LIN {X 0,Y 572.959,Z 403.806,A -85,B 0,C 180,E1 -2247.187,E2 -2247.187} C_VEL
LIN {X 0,Y 572.946,Z 406.184,A -85,B 0,C 180,E1 -2248.594,E2 -2248.594} C_VEL
LIN {X 0,Y 572.938,Z 407,A -85,B 0,C 180,E1 -2249.999,E2 -2249.999} C_VEL
LIN {X 0,Y 572.946,Z 406.187,A -85,B 0,C 180,E1 -2251.405,E2 -2251.405} C_VEL
LIN {X 0,Y 572.959,Z 403.812,A -85,B 0,C 180,E1 -2252.812,E2 -2252.812} C_VEL
LIN {X 0,Y 573.014,Z 400.898,A -85,B 0,C 180,E1 -2253.867,E2 -2253.867} C_VEL
LIN {X 0,Y 572.963,Z 396.952,A -85,B 0,C 180,E1 -2254.925,E2 -2254.925} C_VEL
LIN {X 0,Y 573.093,Z 391.871,A -85,B 0,C 180,E1 -2255.982,E2 -2255.982} C_VEL
LIN {X 0,Y 573.103,Z 385.474,A -85,B 0,C 180,E1 -2257.043,E2 -2257.043} C_VEL
LIN {X 0,Y 573.177,Z 377.485,A -85,B 0,C 180,E1 -2258.105,E2 -2258.105} C_VEL
LIN {X 0,Y 573.253,Z 369.344,A -85,B 0,C 180,E1 -2258.992,E2 -2258.992} C_VEL
LIN {X 0,Y 573.35,Z 359.411,A -85,B 0,C 180,E1 -2259.88,E2 -2259.88} C_VEL
LIN {X 0,Y 573.523,Z 348.2,A -85,B 0,C 180,E1 -2260.68,E2 -2260.68} C_VEL
LIN {X 0,Y 573.627,Z 337.193,A -85,B 0,C 180,E1 -2261.304,E2 -2261.304} C_VEL
LIN {X 0,Y 573.704,Z 325.004,A -85,B 0,C 180,E1 -2261.84,E2 -2261.84} C_VEL
LIN {X 0,Y 573.831,Z 312.213,A -85,B 0,C 180,E1 -2262.241,E2 -2262.241} C_VEL
LIN {X 0,Y 573.922,Z 298.664,A -85,B 0,C 180,E1 -2262.508,E2 -2262.508} C_VEL
LIN {X 0,Y 574.023,Z 199.578,A -85,B 0,C 180,E1 -2263.757,E2 -2263.757} C_VEL
LIN {X 0,Y 573.377,Z 195.275,A -85,B 0,C 180,E1 -2263.85,E2 -2263.85} C_VEL
LIN {X 0,Y 573.52,Z 177.034,A -85,B 0,C 180,E1 -2266.545,E2 -2266.545} C_VEL
LIN {X 0,Y 573.652,Z 159.914,A -85,B 0,C 180,E1 -2269.13,E2 -2269.13} C_VEL
LIN {X 0,Y 573.855,Z 142.746,A -85,B 0,C 180,E1 -2271.744,E2 -2271.744} C_VEL
LIN {X 0,Y 573.214,Z 138.649,A -85,B 0,C 180,E1 -2272.433,E2 -2272.433} C_VEL
LIN {X 0,Y 573.225,Z 138.584,A -85,B 0,C 180,E1 -2275.41,E2 -2275.41} C_VEL
LIN {X 0,Y 573.186,Z 138.585,A -85,B 0,C 180,E1 -2278.016,E2 -2278.016} C_VEL
LIN {X 0,Y 573.201,Z 138.581,A -85,B 0,C 180,E1 -2280.877,E2 -2280.877} C_VEL
LIN {X 0,Y 573.237,Z 138.584,A -85,B 0,C 180,E1 -2283.519,E2 -2283.519} C_VEL
LIN {X 0,Y 573.177,Z 138.584,A -85,B 0,C 180,E1 -2286.053,E2 -2286.053} C_VEL
LIN {X 0,Y 573.17,Z 138.584,A -85,B 0,C 180,E1 -2288.706,E2 -2288.706} C_VEL
LIN {X 0,Y 573.194,Z 138.589,A -85,B 0,C 180,E1 -2291.459,E2 -2291.459} C_VEL
LIN {X 0,Y 573.196,Z 138.58,A -85,B 0,C 180,E1 -2294.335,E2 -2294.335} C_VEL
LIN {X 0,Y 573.189,Z 138.582,A -85,B 0,C 180,E1 -2296.636,E2 -2296.636} C_VEL
LIN {X 0,Y 573.236,Z 138.581,A -85,B 0,C 180,E1 -2299.474,E2 -2299.474} C_VEL
LIN {X 0,Y 573.205,Z 138.578,A -85,B 0,C 180,E1 -2302.19,E2 -2302.19} C_VEL
LIN {X 0,Y 573.215,Z 138.586,A -85,B 0,C 180,E1 -2305.229,E2 -2305.229} C_VEL
LIN {X 0,Y 573.218,Z 138.578,A -85,B 0,C 180,E1 -2307.774,E2 -2307.774} C_VEL
LIN {X 0,Y 573.218,Z 138.58,A -85,B 0,C 180,E1 -2310.631,E2 -2310.631} C_VEL
LIN {X 0,Y 573.189,Z 138.583,A -85,B 0,C 180,E1 -2313.514,E2 -2313.514} C_VEL
LIN {X 0,Y 573.18,Z 138.582,A -85,B 0,C 180,E1 -2316.132,E2 -2316.132} C_VEL
LIN {X 0,Y 573.23,Z 138.581,A -85,B 0,C 180,E1 -2319.173,E2 -2319.173} C_VEL
LIN {X 0,Y 573.189,Z 138.582,A -85,B 0,C 180,E1 -2321.41,E2 -2321.41} C_VEL
LIN {X 0,Y 573.211,Z 138.578,A -85,B 0,C 180,E1 -2323.62,E2 -2323.62} C_VEL
LIN {X 0,Y 573.187,Z 138.586,A -85,B 0,C 180,E1 -2326.528,E2 -2326.528} C_VEL
LIN {X 0,Y 573.221,Z 138.577,A -85,B 0,C 180,E1 -2329.402,E2 -2329.402} C_VEL
LIN {X 0,Y 573.245,Z 138.577,A -85,B 0,C 180,E1 -2332.249,E2 -2332.249} C_VEL
LIN {X 0,Y 573.269,Z 138.574,A -85,B 0,C 180,E1 -2335.077,E2 -2335.077} C_VEL
LIN {X 0,Y 573.27,Z 138.571,A -85,B 0,C 180,E1 -2337.892,E2 -2337.892} C_VEL
LIN {X 0,Y 573.317,Z 138.572,A -85,B 0,C 180,E1 -2340.702,E2 -2340.702} C_VEL
LIN {X 0,Y 573.281,Z 138.574,A -85,B 0,C 180,E1 -2342.81,E2 -2342.81} C_VEL
LIN {X 0,Y 573.246,Z 138.574,A -85,B 0,C 180,E1 -2345.628,E2 -2345.628} C_VEL
LIN {X 0,Y 573.197,Z 138.581,A -85,B 0,C 180,E1 -2347.751,E2 -2347.751} C_VEL
LIN {X 0,Y 573.225,Z 138.583,A -85,B 0,C 180,E1 -2350.597,E2 -2350.597} C_VEL
LIN {X 0,Y 573.194,Z 138.58,A -85,B 0,C 180,E1 -2353.471,E2 -2353.471} C_VEL
LIN {X 0,Y 573.197,Z 138.581,A -85,B 0,C 180,E1 -2355.649,E2 -2355.649} C_VEL
LIN {X 0,Y 573.192,Z 138.584,A -85,B 0,C 180,E1 -2357.85,E2 -2357.85} C_VEL
LIN {X 0,Y 573.218,Z 138.585,A -85,B 0,C 180,E1 -2360.077,E2 -2360.077} C_VEL
LIN {X 0,Y 573.212,Z 138.586,A -85,B 0,C 180,E1 -2362.338,E2 -2362.338} C_VEL
LIN {X 0,Y 573.2,Z 138.581,A -85,B 0,C 180,E1 -2364.394,E2 -2364.394} C_VEL
LIN {X 0,Y 572.557,Z 138.663,A -85,B 0,C 180,E1 -2364.98,E2 -2364.98} C_VEL
LIN {X 0,Y 569.712,Z 139.02,A -85,B 0,C 180,E1 -2365.932,E2 -2365.932} C_VEL
LIN {X 0,Y 567.284,Z 139.319,A -85,B 0,C 180,E1 -2366.697,E2 -2366.697} C_VEL
LIN {X 0,Y 566.228,Z 139.449,A -85,B 0,C 180,E1 -2367.288,E2 -2367.288} C_VEL
LIN {X 0,Y 566.136,Z 139.461,A -85,B 0,C 180,E1 -2367.489,E2 -2367.489} C_VEL
LIN {X 0,Y 566.152,Z 139.462,A -85,B 0,C 180,E1 -2370.594,E2 -2370.594} C_VEL
LIN {X 0,Y 566.246,Z 139.591,A -85,B 0,C 180,E1 -2373.411,E2 -2373.411} C_VEL
LIN {X 0,Y 566.641,Z 143.669,A -85,B 0,C 180,E1 -2374.141,E2 -2374.141} C_VEL
LIN {X 0,Y 566.474,Z 160.639,A -85,B 0,C 180,E1 -2376.988,E2 -2376.988} C_VEL
LIN {X 0,Y 566.291,Z 178.737,A -85,B 0,C 180,E1 -2380,E2 -2380} C_VEL
LIN {X 0,Y 566.525,Z 180.469,A -85,B 0,C 180,E1 -2380.076,E2 -2380.076} C_VEL
LIN {X 0,Y 567.177,Z 186.806,A -85,B 0,C 180,E1 -2380.173,E2 -2380.173} C_VEL
LIN {X 0,Y 566.986,Z 285.959,A -85,B 0,C 180,E1 -2381.451,E2 -2381.451} C_VEL
LIN {X 0,Y 566.852,Z 298.233,A -85,B 0,C 180,E1 -2381.738,E2 -2381.738} C_VEL
LIN {X 0,Y 566.78,Z 308.773,A -85,B 0,C 180,E1 -2382.095,E2 -2382.095} C_VEL
LIN {X 0,Y 566.656,Z 318.628,A -85,B 0,C 180,E1 -2382.527,E2 -2382.527} C_VEL
LIN {X 0,Y 566.545,Z 328.715,A -85,B 0,C 180,E1 -2383.082,E2 -2383.082} C_VEL
LIN {X 0,Y 566.369,Z 338.546,A -85,B 0,C 180,E1 -2383.747,E2 -2383.747} C_VEL
LIN {X 0,Y 566.28,Z 348.816,A -85,B 0,C 180,E1 -2384.598,E2 -2384.598} C_VEL
LIN {X 0,Y 566.11,Z 358.337,A -85,B 0,C 180,E1 -2385.585,E2 -2385.585} C_VEL
LIN {X 0,Y 566.05,Z 365.537,A -85,B 0,C 180,E1 -2386.497,E2 -2386.497} C_VEL
LIN {X 0,Y 565.975,Z 372.063,A -85,B 0,C 180,E1 -2387.498,E2 -2387.498} C_VEL
LIN {X 0,Y 565.954,Z 377.399,A -85,B 0,C 180,E1 -2388.503,E2 -2388.503} C_VEL
LIN {X 0,Y 565.92,Z 382.712,A -85,B 0,C 180,E1 -2389.778,E2 -2389.778} C_VEL
LIN {X 0,Y 565.842,Z 385.534,A -85,B 0,C 180,E1 -2390.697,E2 -2390.697} C_VEL
LIN {X 0,Y 565.844,Z 387.622,A -85,B 0,C 180,E1 -2391.611,E2 -2391.611} C_VEL
LIN {X 0,Y 565.828,Z 389.187,A -85,B 0,C 180,E1 -2392.648,E2 -2392.648} C_VEL
LIN {X 0,Y 565.813,Z 389.96,A -85,B 0,C 180,E1 -2393.839,E2 -2393.839} C_VEL
LIN {X 0,Y 565.849,Z 389.512,A -85,B 0,C 180,E1 -2395.158,E2 -2395.158} C_VEL
LIN {X 0,Y 565.86,Z 387.946,A -85,B 0,C 180,E1 -2396.319,E2 -2396.319} C_VEL
LIN {X 0,Y 565.883,Z 384.566,A -85,B 0,C 180,E1 -2397.723,E2 -2397.723} C_VEL
LIN {X 0,Y 565.936,Z 381.748,A -85,B 0,C 180,E1 -2398.564,E2 -2398.564} C_VEL
LIN {X 0,Y 565.945,Z 376.347,A -85,B 0,C 180,E1 -2399.807,E2 -2399.807} C_VEL
LIN {X 0,Y 566.013,Z 369.386,A -85,B 0,C 180,E1 -2401.038,E2 -2401.038} C_VEL
LIN {X 0,Y 566.097,Z 362.063,A -85,B 0,C 180,E1 -2402.054,E2 -2402.054} C_VEL
LIN {X 0,Y 566.182,Z 355.241,A -85,B 0,C 180,E1 -2402.847,E2 -2402.847} C_VEL
LIN {X 0,Y 566.273,Z 346.877,A -85,B 0,C 180,E1 -2403.662,E2 -2403.662} C_VEL
LIN {X 0,Y 566.371,Z 338.436,A -85,B 0,C 180,E1 -2404.351,E2 -2404.351} C_VEL
LIN {X 0,Y 566.495,Z 329.013,A -85,B 0,C 180,E1 -2404.99,E2 -2404.99} C_VEL
LIN {X 0,Y 566.641,Z 318.934,A -85,B 0,C 180,E1 -2405.548,E2 -2405.548} C_VEL
LIN {X 0,Y 566.78,Z 307.631,A -85,B 0,C 180,E1 -2406.042,E2 -2406.042} C_VEL
LIN {X 0,Y 566.903,Z 293.652,A -85,B 0,C 180,E1 -2406.476,E2 -2406.476} C_VEL
LIN {X 0,Y 566.983,Z 281.874,A -85,B 0,C 180,E1 -2406.705,E2 -2406.705} C_VEL
LIN {X 0,Y 567.054,Z 183.818,A -85,B 0,C 180,E1 -2407.958,E2 -2407.958} C_VEL
LIN {X 0,Y 566.338,Z 179.288,A -85,B 0,C 180,E1 -2408.049,E2 -2408.049} C_VEL
LIN {X 0,Y 566.292,Z 178.336,A -85,B 0,C 180,E1 -2408.143,E2 -2408.143} C_VEL
LIN {X 0,Y 566.417,Z 162.116,A -85,B 0,C 180,E1 -2410.872,E2 -2410.872} C_VEL
LIN {X 0,Y 566.688,Z 143.921,A -85,B 0,C 180,E1 -2413.983,E2 -2413.983} C_VEL
LIN {X 0,Y 566.248,Z 139.507,A -85,B 0,C 180,E1 -2414.801,E2 -2414.801} C_VEL
LIN {X 0,Y 566.24,Z 139.454,A -85,B 0,C 180,E1 -2417.82,E2 -2417.82} C_VEL
LIN {X 0,Y 566.209,Z 139.451,A -85,B 0,C 180,E1 -2420.715,E2 -2420.715} C_VEL
LIN {X 0,Y 566.262,Z 139.444,A -85,B 0,C 180,E1 -2423.164,E2 -2423.164} C_VEL
LIN {X 0,Y 566.182,Z 139.461,A -85,B 0,C 180,E1 -2425.73,E2 -2425.73} C_VEL
LIN {X 0,Y 566.275,Z 139.451,A -85,B 0,C 180,E1 -2427.867,E2 -2427.867} C_VEL
LIN {X 0,Y 566.298,Z 139.439,A -85,B 0,C 180,E1 -2430.712,E2 -2430.712} C_VEL
LIN {X 0,Y 566.268,Z 139.443,A -85,B 0,C 180,E1 -2432.846,E2 -2432.846} C_VEL
LIN {X 0,Y 566.254,Z 139.453,A -85,B 0,C 180,E1 -2435.699,E2 -2435.699} C_VEL
LIN {X 0,Y 566.204,Z 139.451,A -85,B 0,C 180,E1 -2438.567,E2 -2438.567} C_VEL
LIN {X 0,Y 566.241,Z 139.455,A -85,B 0,C 180,E1 -2441.455,E2 -2441.455} C_VEL
LIN {X 0,Y 566.228,Z 139.448,A -85,B 0,C 180,E1 -2444.505,E2 -2444.505} C_VEL
LIN {X 0,Y 566.198,Z 139.461,A -85,B 0,C 180,E1 -2447.332,E2 -2447.332} C_VEL
LIN {X 0,Y 566.206,Z 139.45,A -85,B 0,C 180,E1 -2450.338,E2 -2450.338} C_VEL
LIN {X 0,Y 566.17,Z 139.464,A -85,B 0,C 180,E1 -2453.282,E2 -2453.282} C_VEL
LIN {X 0,Y 566.207,Z 139.452,A -85,B 0,C 180,E1 -2455.75,E2 -2455.75} C_VEL
LIN {X 0,Y 566.202,Z 139.451,A -85,B 0,C 180,E1 -2458.202,E2 -2458.202} C_VEL
LIN {X 0,Y 566.185,Z 139.463,A -85,B 0,C 180,E1 -2461.076,E2 -2461.076} C_VEL
LIN {X 0,Y 566.196,Z 139.452,A -85,B 0,C 180,E1 -2463.732,E2 -2463.732} C_VEL
LIN {X 0,Y 566.198,Z 139.455,A -85,B 0,C 180,E1 -2466.57,E2 -2466.57} C_VEL
LIN {X 0,Y 566.211,Z 139.45,A -85,B 0,C 180,E1 -2469.686,E2 -2469.686} C_VEL
LIN {X 0,Y 566.197,Z 139.46,A -85,B 0,C 180,E1 -2472.917,E2 -2472.917} C_VEL
LIN {X 0,Y 566.192,Z 139.453,A -85,B 0,C 180,E1 -2476.05,E2 -2476.05} C_VEL
LIN {X 0,Y 566.201,Z 139.453,A -85,B 0,C 180,E1 -2479.215,E2 -2479.215} C_VEL
LIN {X 0,Y 566.179,Z 139.454,A -85,B 0,C 180,E1 -2481.637,E2 -2481.637} C_VEL
LIN {X 0,Y 566.147,Z 139.463,A -85,B 0,C 180,E1 -2484.307,E2 -2484.307} C_VEL
LIN {X 0,Y 566.217,Z 139.453,A -85,B 0,C 180,E1 -2486.898,E2 -2486.898} C_VEL
LIN {X 0,Y 566.174,Z 139.454,A -85,B 0,C 180,E1 -2489.407,E2 -2489.407} C_VEL
LIN {X 0,Y 566.185,Z 139.455,A -85,B 0,C 180,E1 -2491.856,E2 -2491.856} C_VEL
LIN {X 0,Y 566.236,Z 139.447,A -85,B 0,C 180,E1 -2495.039,E2 -2495.039} C_VEL
LIN {X 0,Y 566.184,Z 139.461,A -85,B 0,C 180,E1 -2498.137,E2 -2498.137} C_VEL
LIN {X 0,Y 566.229,Z 139.451,A -85,B 0,C 180,E1 -2500.614,E2 -2500.614} C_VEL
LIN {X 0,Y 566.176,Z 139.455,A -85,B 0,C 180,E1 -2503.412,E2 -2503.412} C_VEL
LIN {X 0,Y 566.181,Z 139.459,A -85,B 0,C 180,E1 -2506.359,E2 -2506.359} C_VEL
LIN {X 0,Y 566.234,Z 139.448,A -85,B 0,C 180,E1 -2508.676,E2 -2508.676} C_VEL
LIN {X 0,Y 566.198,Z 139.454,A -85,B 0,C 180,E1 -2511.434,E2 -2511.434} C_VEL
LIN {X 0,Y 566.235,Z 139.45,A -85,B 0,C 180,E1 -2514.302,E2 -2514.302} C_VEL
LIN {X 0,Y 566.271,Z 139.452,A -85,B 0,C 180,E1 -2517.867,E2 -2517.867} C_VEL
LIN {X 0,Y 566.279,Z 139.448,A -85,B 0,C 180,E1 -2520,E2 -2520} C_VEL
LIN {X 0,Y 566.249,Z 139.445,A -85,B 0,C 180,E1 -2522.846,E2 -2522.846} C_VEL
LIN {X 0,Y 566.24,Z 139.456,A -85,B 0,C 180,E1 -2525.699,E2 -2525.699} C_VEL
LIN {X 0,Y 566.187,Z 139.453,A -85,B 0,C 180,E1 -2528.567,E2 -2528.567} C_VEL
LIN {X 0,Y 566.238,Z 139.455,A -85,B 0,C 180,E1 -2531.455,E2 -2531.455} C_VEL
LIN {X 0,Y 566.176,Z 139.454,A -85,B 0,C 180,E1 -2534.483,E2 -2534.483} C_VEL
LIN {X 0,Y 566.181,Z 139.462,A -85,B 0,C 180,E1 -2537.333,E2 -2537.333} C_VEL
LIN {X 0,Y 566.196,Z 139.458,A -85,B 0,C 180,E1 -2539.581,E2 -2539.581} C_VEL
LIN {X 0,Y 566.181,Z 139.455,A -85,B 0,C 180,E1 -2541.863,E2 -2541.863} C_VEL
LIN {X 0,Y 566.152,Z 139.457,A -85,B 0,C 180,E1 -2544.183,E2 -2544.183} C_VEL
LIN {X 0,Y 566.166,Z 139.457,A -85,B 0,C 180,E1 -2546.651,E2 -2546.651} C_VEL
LIN {X 0,Y 566.146,Z 139.459,A -85,B 0,C 180,E1 -2549.772,E2 -2549.772} C_VEL
LIN {X 0,Y 566.176,Z 139.455,A -85,B 0,C 180,E1 -2552.425,E2 -2552.425} C_VEL
LIN {X 0,Y 566.164,Z 139.465,A -85,B 0,C 180,E1 -2554.987,E2 -2554.987} C_VEL
LIN {X 0,Y 566.185,Z 139.456,A -85,B 0,C 180,E1 -2557.462,E2 -2557.462} C_VEL
LIN {X 0,Y 566.159,Z 139.457,A -85,B 0,C 180,E1 -2560.204,E2 -2560.204} C_VEL
LIN {X 0,Y 566.144,Z 139.464,A -85,B 0,C 180,E1 -2563.06,E2 -2563.06} C_VEL
LIN {X 0,Y 566.144,Z 139.459,A -85,B 0,C 180,E1 -2566.055,E2 -2566.055} C_VEL
LIN {X 0,Y 566.138,Z 139.466,A -85,B 0,C 180,E1 -2568.857,E2 -2568.857} C_VEL
LIN {X 0,Y 566.13,Z 139.46,A -85,B 0,C 180,E1 -2571.453,E2 -2571.453} C_VEL
LIN {X 0,Y 566.152,Z 139.457,A -85,B 0,C 180,E1 -2573.793,E2 -2573.793} C_VEL
LIN {X 0,Y 566.143,Z 139.462,A -85,B 0,C 180,E1 -2576.892,E2 -2576.892} C_VEL
LIN {X 0,Y 566.149,Z 139.458,A -85,B 0,C 180,E1 -2579.405,E2 -2579.405} C_VEL
LIN {X 0,Y 566.133,Z 139.462,A -85,B 0,C 180,E1 -2581.853,E2 -2581.853} C_VEL
LIN {X 0,Y 566.178,Z 139.462,A -85,B 0,C 180,E1 -2584.249,E2 -2584.249} C_VEL
LIN {X 0,Y 566.178,Z 139.567,A -85,B 0,C 180,E1 -2587.416,E2 -2587.416} C_VEL
LIN {X 0,Y 566.945,Z 143.998,A -85,B 0,C 180,E1 -2588.167,E2 -2588.167} C_VEL
LIN {X 0,Y 566.702,Z 161.238,A -85,B 0,C 180,E1 -2590.837,E2 -2590.837} C_VEL
LIN {X 0,Y 566.514,Z 177.105,A -85,B 0,C 180,E1 -2593.261,E2 -2593.261} C_VEL
LIN {X 0,Y 566.384,Z 195.262,A -85,B 0,C 180,E1 -2595.974,E2 -2595.974} C_VEL
LIN {X 0,Y 567.129,Z 200.463,A -85,B 0,C 180,E1 -2596.084,E2 -2596.084} C_VEL
LIN {X 0,Y 566.982,Z 302.917,A -85,B 0,C 180,E1 -2597.403,E2 -2597.403} C_VEL
LIN {X 0,Y 566.858,Z 316.198,A -85,B 0,C 180,E1 -2597.718,E2 -2597.718} C_VEL
LIN {X 0,Y 566.73,Z 328.363,A -85,B 0,C 180,E1 -2598.147,E2 -2598.147} C_VEL
LIN {X 0,Y 566.629,Z 340.142,A -85,B 0,C 180,E1 -2598.708,E2 -2598.708} C_VEL
LIN {X 0,Y 566.461,Z 352.187,A -85,B 0,C 180,E1 -2599.455,E2 -2599.455} C_VEL
LIN {X 0,Y 566.326,Z 362.597,A -85,B 0,C 180,E1 -2600.265,E2 -2600.265} C_VEL
LIN {X 0,Y 566.207,Z 371.107,A -85,B 0,C 180,E1 -2601.074,E2 -2601.074} C_VEL
LIN {X 0,Y 566.113,Z 378.955,A -85,B 0,C 180,E1 -2601.971,E2 -2601.971} C_VEL
LIN {X 0,Y 566.004,Z 386.619,A -85,B 0,C 180,E1 -2603.046,E2 -2603.046} C_VEL
LIN {X 0,Y 566.004,Z 393.676,A -85,B 0,C 180,E1 -2604.298,E2 -2604.298} C_VEL
LIN {X 0,Y 565.933,Z 398.37,A -85,B 0,C 180,E1 -2605.369,E2 -2605.369} C_VEL
LIN {X 0,Y 565.927,Z 401.956,A -85,B 0,C 180,E1 -2606.439,E2 -2606.439} C_VEL
LIN {X 0,Y 565.878,Z 403.806,A -85,B 0,C 180,E1 -2607.152,E2 -2607.152} C_VEL
LIN {X 0,Y 565.846,Z 406.183,A -85,B 0,C 180,E1 -2608.576,E2 -2608.576} C_VEL
LIN {X 0,Y 565.839,Z 407,A -85,B 0,C 180,E1 -2609.999,E2 -2609.999} C_VEL
LIN {X 0,Y 565.846,Z 406.186,A -85,B 0,C 180,E1 -2611.423,E2 -2611.423} C_VEL
LIN {X 0,Y 565.878,Z 403.812,A -85,B 0,C 180,E1 -2612.847,E2 -2612.847} C_VEL
LIN {X 0,Y 565.926,Z 400.898,A -85,B 0,C 180,E1 -2613.916,E2 -2613.916} C_VEL
LIN {X 0,Y 565.878,Z 396.952,A -85,B 0,C 180,E1 -2614.987,E2 -2614.987} C_VEL
LIN {X 0,Y 566.004,Z 391.872,A -85,B 0,C 180,E1 -2616.058,E2 -2616.058} C_VEL
LIN {X 0,Y 566.039,Z 385.473,A -85,B 0,C 180,E1 -2617.131,E2 -2617.131} C_VEL
LIN {X 0,Y 566.133,Z 377.485,A -85,B 0,C 180,E1 -2618.207,E2 -2618.207} C_VEL
LIN {X 0,Y 566.228,Z 369.343,A -85,B 0,C 180,E1 -2619.105,E2 -2619.105} C_VEL
LIN {X 0,Y 566.351,Z 359.409,A -85,B 0,C 180,E1 -2620.004,E2 -2620.004} C_VEL
LIN {X 0,Y 566.544,Z 348.298,A -85,B 0,C 180,E1 -2620.806,E2 -2620.806} C_VEL
LIN {X 0,Y 566.659,Z 337.191,A -85,B 0,C 180,E1 -2621.445,E2 -2621.445} C_VEL
LIN {X 0,Y 566.743,Z 325.002,A -85,B 0,C 180,E1 -2621.987,E2 -2621.987} C_VEL
LIN {X 0,Y 566.907,Z 312.212,A -85,B 0,C 180,E1 -2622.393,E2 -2622.393} C_VEL
LIN {X 0,Y 567,Z 300.167,A -85,B 0,C 180,E1 -2622.641,E2 -2622.641} C_VEL
LIN {X 0,Y 567.039,Z 199.902,A -85,B 0,C 180,E1 -2623.925,E2 -2623.925} C_VEL
LIN {X 0,Y 566.37,Z 195.286,A -85,B 0,C 180,E1 -2624.025,E2 -2624.025} C_VEL
LIN {X 0,Y 566.53,Z 176.033,A -85,B 0,C 180,E1 -2626.896,E2 -2626.896} C_VEL
LIN {X 0,Y 566.715,Z 158.543,A -85,B 0,C 180,E1 -2629.561,E2 -2629.561} C_VEL
LIN {X 0,Y 566.892,Z 143.82,A -85,B 0,C 180,E1 -2631.833,E2 -2631.833} C_VEL
LIN {X 0,Y 566.189,Z 139.553,A -85,B 0,C 180,E1 -2632.558,E2 -2632.558} C_VEL
LIN {X 0,Y 566.186,Z 139.462,A -85,B 0,C 180,E1 -2635.749,E2 -2635.749} C_VEL
LIN {X 0,Y 566.131,Z 139.463,A -85,B 0,C 180,E1 -2638.188,E2 -2638.188} C_VEL
LIN {X 0,Y 566.17,Z 139.459,A -85,B 0,C 180,E1 -2641.072,E2 -2641.072} C_VEL
LIN {X 0,Y 566.19,Z 139.459,A -85,B 0,C 180,E1 -2643.73,E2 -2643.73} C_VEL
LIN {X 0,Y 566.137,Z 139.46,A -85,B 0,C 180,E1 -2646.573,E2 -2646.573} C_VEL
LIN {X 0,Y 566.192,Z 139.458,A -85,B 0,C 180,E1 -2649.683,E2 -2649.683} C_VEL
LIN {X 0,Y 566.141,Z 139.462,A -85,B 0,C 180,E1 -2652.91,E2 -2652.91} C_VEL
LIN {X 0,Y 566.144,Z 139.459,A -85,B 0,C 180,E1 -2656.053,E2 -2656.053} C_VEL
LIN {X 0,Y 566.144,Z 139.462,A -85,B 0,C 180,E1 -2658.857,E2 -2658.857} C_VEL
LIN {X 0,Y 566.188,Z 139.458,A -85,B 0,C 180,E1 -2661.443,E2 -2661.443} C_VEL
LIN {X 0,Y 566.132,Z 139.46,A -85,B 0,C 180,E1 -2664.305,E2 -2664.305} C_VEL
LIN {X 0,Y 566.15,Z 139.463,A -85,B 0,C 180,E1 -2666.893,E2 -2666.893} C_VEL
LIN {X 0,Y 566.147,Z 139.462,A -85,B 0,C 180,E1 -2669.405,E2 -2669.405} C_VEL
LIN {X 0,Y 566.138,Z 139.459,A -85,B 0,C 180,E1 -2671.853,E2 -2671.853} C_VEL
LIN {X 0,Y 566.169,Z 139.456,A -85,B 0,C 180,E1 -2674.249,E2 -2674.249} C_VEL
LIN {X 0,Y 566.146,Z 139.461,A -85,B 0,C 180,E1 -2677.367,E2 -2677.367} C_VEL
LIN {X 0,Y 566.185,Z 139.453,A -85,B 0,C 180,E1 -2679.661,E2 -2679.661} C_VEL
LIN {X 0,Y 566.161,Z 139.456,A -85,B 0,C 180,E1 -2681.92,E2 -2681.92} C_VEL
LIN {X 0,Y 566.169,Z 139.463,A -85,B 0,C 180,E1 -2684.889,E2 -2684.889} C_VEL
LIN {X 0,Y 566.163,Z 139.456,A -85,B 0,C 180,E1 -2687.817,E2 -2687.817} C_VEL
LIN {X 0,Y 566.141,Z 139.459,A -85,B 0,C 180,E1 -2689.991,E2 -2689.991} C_VEL
LIN {X 0,Y 566.225,Z 139.454,A -85,B 0,C 180,E1 -2692.87,E2 -2692.87} C_VEL
LIN {X 0,Y 566.245,Z 139.449,A -85,B 0,C 180,E1 -2695.015,E2 -2695.015} C_VEL
LIN {X 0,Y 566.244,Z 139.446,A -85,B 0,C 180,E1 -2697.866,E2 -2697.866} C_VEL
LIN {X 0,Y 566.286,Z 139.448,A -85,B 0,C 180,E1 -2700.711,E2 -2700.711} C_VEL
LIN {X 0,Y 566.245,Z 139.449,A -85,B 0,C 180,E1 -2702.845,E2 -2702.845} C_VEL
LIN {X 0,Y 566.217,Z 139.45,A -85,B 0,C 180,E1 -2705.698,E2 -2705.698} C_VEL
LIN {X 0,Y 566.168,Z 139.457,A -85,B 0,C 180,E1 -2707.848,E2 -2707.848} C_VEL
LIN {X 0,Y 566.195,Z 139.456,A -85,B 0,C 180,E1 -2710.73,E2 -2710.73} C_VEL
LIN {X 0,Y 566.163,Z 139.458,A -85,B 0,C 180,E1 -2712.911,E2 -2712.911} C_VEL
LIN {X 0,Y 566.17,Z 139.456,A -85,B 0,C 180,E1 -2715.11,E2 -2715.11} C_VEL
LIN {X 0,Y 566.153,Z 139.464,A -85,B 0,C 180,E1 -2718.079,E2 -2718.079} C_VEL
LIN {X 0,Y 566.186,Z 139.461,A -85,B 0,C 180,E1 -2720.338,E2 -2720.338} C_VEL
LIN {X 0,Y 566.151,Z 139.458,A -85,B 0,C 180,E1 -2723.28,E2 -2723.28} C_VEL
LIN {X 0,Y 566.172,Z 139.459,A -85,B 0,C 180,E1 -2725.751,E2 -2725.751} C_VEL
LIN {X 0,Y 566.136,Z 139.461,A -85,B 0,C 180,E1 -2727.489,E2 -2727.489} C_VEL
LIN {X 0,Y 565.452,Z 139.554,A -85,B 0,C 180,E1 -2728.082,E2 -2728.082} C_VEL
LIN {X 0,Y 562.596,Z 139.908,A -85,B 0,C 180,E1 -2729.046,E2 -2729.046} C_VEL
LIN {X 0,Y 560.202,Z 140.206,A -85,B 0,C 180,E1 -2729.822,E2 -2729.822} C_VEL
LIN {X 0,Y 559.187,Z 140.332,A -85,B 0,C 180,E1 -2730.421,E2 -2730.421} C_VEL
LIN {X 0,Y 559.11,Z 140.338,A -85,B 0,C 180,E1 -2730.624,E2 -2730.624} C_VEL
LIN {X 0,Y 559.184,Z 140.438,A -85,B 0,C 180,E1 -2733.303,E2 -2733.303} C_VEL
LIN {X 0,Y 559.641,Z 144.369,A -85,B 0,C 180,E1 -2734.024,E2 -2734.024} C_VEL
LIN {X 0,Y 559.477,Z 160.467,A -85,B 0,C 180,E1 -2736.754,E2 -2736.754} C_VEL
LIN {X 0,Y 559.283,Z 179.019,A -85,B 0,C 180,E1 -2739.842,E2 -2739.842} C_VEL
LIN {X 0,Y 560.263,Z 185.188,A -85,B 0,C 180,E1 -2739.977,E2 -2739.977} C_VEL
LIN {X 0,Y 560.037,Z 285.586,A -85,B 0,C 180,E1 -2741.287,E2 -2741.287} C_VEL
LIN {X 0,Y 559.926,Z 298.604,A -85,B 0,C 180,E1 -2741.596,E2 -2741.596} C_VEL
LIN {X 0,Y 559.811,Z 309.088,A -85,B 0,C 180,E1 -2741.958,E2 -2741.958} C_VEL
LIN {X 0,Y 559.732,Z 317.871,A -85,B 0,C 180,E1 -2742.345,E2 -2742.345} C_VEL
LIN {X 0,Y 559.578,Z 327.966,A -85,B 0,C 180,E1 -2742.898,E2 -2742.898} C_VEL
LIN {X 0,Y 559.404,Z 336.205,A -85,B 0,C 180,E1 -2743.444,E2 -2743.444} C_VEL
LIN {X 0,Y 559.304,Z 344.724,A -85,B 0,C 180,E1 -2744.119,E2 -2744.119} C_VEL
LIN {X 0,Y 559.162,Z 352.208,A -85,B 0,C 180,E1 -2744.817,E2 -2744.817} C_VEL
LIN {X 0,Y 559.061,Z 358.864,A -85,B 0,C 180,E1 -2745.544,E2 -2745.544} C_VEL
LIN {X 0,Y 558.986,Z 365.585,A -85,B 0,C 180,E1 -2746.41,E2 -2746.41} C_VEL
LIN {X 0,Y 558.891,Z 372.031,A -85,B 0,C 180,E1 -2747.411,E2 -2747.411} C_VEL
LIN {X 0,Y 558.879,Z 376.314,A -85,B 0,C 180,E1 -2748.206,E2 -2748.206} C_VEL
LIN {X 0,Y 558.84,Z 380.573,A -85,B 0,C 180,E1 -2749.161,E2 -2749.161} C_VEL
LIN {X 0,Y 558.792,Z 383.93,A -85,B 0,C 180,E1 -2750.103,E2 -2750.103} C_VEL
LIN {X 0,Y 558.743,Z 386.933,A -85,B 0,C 180,E1 -2751.246,E2 -2751.246} C_VEL
LIN {X 0,Y 558.736,Z 388.915,A -85,B 0,C 180,E1 -2752.413,E2 -2752.413} C_VEL
LIN {X 0,Y 558.724,Z 389.862,A -85,B 0,C 180,E1 -2753.613,E2 -2753.613} C_VEL
LIN {X 0,Y 558.749,Z 389.714,A -85,B 0,C 180,E1 -2754.842,E2 -2754.842} C_VEL
LIN {X 0,Y 558.764,Z 388.361,A -85,B 0,C 180,E1 -2756.112,E2 -2756.112} C_VEL
LIN {X 0,Y 558.774,Z 385.553,A -85,B 0,C 180,E1 -2757.425,E2 -2757.425} C_VEL
LIN {X 0,Y 558.834,Z 382.284,A -85,B 0,C 180,E1 -2758.477,E2 -2758.477} C_VEL
LIN {X 0,Y 558.863,Z 378.689,A -85,B 0,C 180,E1 -2759.384,E2 -2759.384} C_VEL
LIN {X 0,Y 558.946,Z 373.565,A -85,B 0,C 180,E1 -2760.412,E2 -2760.412} C_VEL
LIN {X 0,Y 558.969,Z 368.511,A -85,B 0,C 180,E1 -2761.256,E2 -2761.256} C_VEL
LIN {X 0,Y 559.039,Z 361.027,A -85,B 0,C 180,E1 -2762.282,E2 -2762.282} C_VEL
LIN {X 0,Y 559.176,Z 353.184,A -85,B 0,C 180,E1 -2763.171,E2 -2763.171} C_VEL
LIN {X 0,Y 559.27,Z 345.44,A -85,B 0,C 180,E1 -2763.909,E2 -2763.909} C_VEL
LIN {X 0,Y 559.438,Z 336.59,A -85,B 0,C 180,E1 -2764.616,E2 -2764.616} C_VEL
LIN {X 0,Y 559.577,Z 325.942,A -85,B 0,C 180,E1 -2765.318,E2 -2765.318} C_VEL
LIN {X 0,Y 559.747,Z 313.14,A -85,B 0,C 180,E1 -2765.967,E2 -2765.967} C_VEL
LIN {X 0,Y 559.893,Z 301.825,A -85,B 0,C 180,E1 -2766.394,E2 -2766.394} C_VEL
LIN {X 0,Y 560,Z 290.948,A -85,B 0,C 180,E1 -2766.694,E2 -2766.694} C_VEL
LIN {X 0,Y 560.09,Z 276.268,A -85,B 0,C 180,E1 -2766.94,E2 -2766.94} C_VEL
LIN {X 0,Y 560.193,Z 184.677,A -85,B 0,C 180,E1 -2768.122,E2 -2768.122} C_VEL
LIN {X 0,Y 559.307,Z 179.219,A -85,B 0,C 180,E1 -2768.235,E2 -2768.235} C_VEL
LIN {X 0,Y 559.242,Z 176.579,A -85,B 0,C 180,E1 -2768.628,E2 -2768.628} C_VEL
LIN {X 0,Y 559.475,Z 160.858,A -85,B 0,C 180,E1 -2771.319,E2 -2771.319} C_VEL
LIN {X 0,Y 559.724,Z 144.461,A -85,B 0,C 180,E1 -2774.152,E2 -2774.152} C_VEL
LIN {X 0,Y 559.2,Z 140.378,A -85,B 0,C 180,E1 -2774.929,E2 -2774.929} C_VEL
LIN {X 0,Y 559.194,Z 140.33,A -85,B 0,C 180,E1 -2777.664,E2 -2777.664} C_VEL
LIN {X 0,Y 559.181,Z 140.327,A -85,B 0,C 180,E1 -2780.597,E2 -2780.597} C_VEL
LIN {X 0,Y 559.223,Z 140.321,A -85,B 0,C 180,E1 -2783.13,E2 -2783.13} C_VEL
LIN {X 0,Y 559.142,Z 140.337,A -85,B 0,C 180,E1 -2785.676,E2 -2785.676} C_VEL
LIN {X 0,Y 559.247,Z 140.326,A -85,B 0,C 180,E1 -2787.84,E2 -2787.84} C_VEL
LIN {X 0,Y 559.268,Z 140.315,A -85,B 0,C 180,E1 -2790.721,E2 -2790.721} C_VEL
LIN {X 0,Y 559.235,Z 140.319,A -85,B 0,C 180,E1 -2792.882,E2 -2792.882} C_VEL
LIN {X 0,Y 559.224,Z 140.327,A -85,B 0,C 180,E1 -2795.771,E2 -2795.771} C_VEL
LIN {X 0,Y 559.168,Z 140.327,A -85,B 0,C 180,E1 -2798.675,E2 -2798.675} C_VEL
LIN {X 0,Y 559.204,Z 140.331,A -85,B 0,C 180,E1 -2801.601,E2 -2801.601} C_VEL
LIN {X 0,Y 559.199,Z 140.323,A -85,B 0,C 180,E1 -2804.596,E2 -2804.596} C_VEL
LIN {X 0,Y 559.141,Z 140.337,A -85,B 0,C 180,E1 -2807.558,E2 -2807.558} C_VEL
LIN {X 0,Y 559.164,Z 140.33,A -85,B 0,C 180,E1 -2809.838,E2 -2809.838} C_VEL
LIN {X 0,Y 559.139,Z 140.331,A -85,B 0,C 180,E1 -2812.153,E2 -2812.153} C_VEL
LIN {X 0,Y 559.174,Z 140.334,A -85,B 0,C 180,E1 -2815.299,E2 -2815.299} C_VEL
LIN {X 0,Y 559.156,Z 140.33,A -85,B 0,C 180,E1 -2817.714,E2 -2817.714} C_VEL
LIN {X 0,Y 559.146,Z 140.33,A -85,B 0,C 180,E1 -2820.184,E2 -2820.184} C_VEL
LIN {X 0,Y 559.152,Z 140.334,A -85,B 0,C 180,E1 -2822.716,E2 -2822.716} C_VEL
LIN {X 0,Y 559.126,Z 140.337,A -85,B 0,C 180,E1 -2825.324,E2 -2825.324} C_VEL
LIN {X 0,Y 559.13,Z 140.332,A -85,B 0,C 180,E1 -2828.018,E2 -2828.018} C_VEL
LIN {X 0,Y 559.154,Z 140.338,A -85,B 0,C 180,E1 -2830.813,E2 -2830.813} C_VEL
LIN {X 0,Y 559.135,Z 140.331,A -85,B 0,C 180,E1 -2833.735,E2 -2833.735} C_VEL
LIN {X 0,Y 559.14,Z 140.339,A -85,B 0,C 180,E1 -2836.804,E2 -2836.804} C_VEL
LIN {X 0,Y 559.153,Z 140.331,A -85,B 0,C 180,E1 -2839.188,E2 -2839.188} C_VEL
LIN {X 0,Y 559.127,Z 140.334,A -85,B 0,C 180,E1 -2841.982,E2 -2841.982} C_VEL
LIN {X 0,Y 559.126,Z 140.338,A -85,B 0,C 180,E1 -2844.788,E2 -2844.788} C_VEL
LIN {X 0,Y 559.153,Z 140.329,A -85,B 0,C 180,E1 -2847.365,E2 -2847.365} C_VEL
LIN {X 0,Y 559.144,Z 140.335,A -85,B 0,C 180,E1 -2850.143,E2 -2850.143} C_VEL
LIN {X 0,Y 559.139,Z 140.331,A -85,B 0,C 180,E1 -2853.179,E2 -2853.179} C_VEL
LIN {X 0,Y 559.154,Z 140.329,A -85,B 0,C 180,E1 -2855.495,E2 -2855.495} C_VEL
LIN {X 0,Y 559.169,Z 140.331,A -85,B 0,C 180,E1 -2858.624,E2 -2858.624} C_VEL
LIN {X 0,Y 559.156,Z 140.329,A -85,B 0,C 180,E1 -2860.926,E2 -2860.926} C_VEL
LIN {X 0,Y 559.142,Z 140.337,A -85,B 0,C 180,E1 -2863.948,E2 -2863.948} C_VEL
LIN {X 0,Y 559.157,Z 140.337,A -85,B 0,C 180,E1 -2866.184,E2 -2866.184} C_VEL
LIN {X 0,Y 559.189,Z 140.325,A -85,B 0,C 180,E1 -2869.134,E2 -2869.134} C_VEL
LIN {X 0,Y 559.169,Z 140.335,A -85,B 0,C 180,E1 -2872.053,E2 -2872.053} C_VEL
LIN {X 0,Y 559.237,Z 140.318,A -85,B 0,C 180,E1 -2874.954,E2 -2874.954} C_VEL
LIN {X 0,Y 559.242,Z 140.328,A -85,B 0,C 180,E1 -2877.84,E2 -2877.84} C_VEL
LIN {X 0,Y 559.248,Z 140.323,A -85,B 0,C 180,E1 -2880,E2 -2880} C_VEL
LIN {X 0,Y 559.218,Z 140.321,A -85,B 0,C 180,E1 -2882.882,E2 -2882.882} C_VEL
LIN {X 0,Y 559.206,Z 140.33,A -85,B 0,C 180,E1 -2885.771,E2 -2885.771} C_VEL
LIN {X 0,Y 559.153,Z 140.329,A -85,B 0,C 180,E1 -2888.675,E2 -2888.675} C_VEL
LIN {X 0,Y 559.196,Z 140.332,A -85,B 0,C 180,E1 -2891.601,E2 -2891.601} C_VEL
LIN {X 0,Y 559.152,Z 140.329,A -85,B 0,C 180,E1 -2894.576,E2 -2894.576} C_VEL
LIN {X 0,Y 559.127,Z 140.339,A -85,B 0,C 180,E1 -2897.558,E2 -2897.558} C_VEL
LIN {X 0,Y 559.152,Z 140.332,A -85,B 0,C 180,E1 -2899.838,E2 -2899.838} C_VEL
LIN {X 0,Y 559.128,Z 140.332,A -85,B 0,C 180,E1 -2902.154,E2 -2902.154} C_VEL
LIN {X 0,Y 559.129,Z 140.341,A -85,B 0,C 180,E1 -2905.176,E2 -2905.176} C_VEL
LIN {X 0,Y 559.101,Z 140.338,A -85,B 0,C 180,E1 -2907.717,E2 -2907.717} C_VEL
LIN {X 0,Y 559.092,Z 140.337,A -85,B 0,C 180,E1 -2910.187,E2 -2910.187} C_VEL
LIN {X 0,Y 559.134,Z 140.335,A -85,B 0,C 180,E1 -2912.717,E2 -2912.717} C_VEL
LIN {X 0,Y 559.115,Z 140.339,A -85,B 0,C 180,E1 -2915.325,E2 -2915.325} C_VEL
LIN {X 0,Y 559.122,Z 140.333,A -85,B 0,C 180,E1 -2918.019,E2 -2918.019} C_VEL
LIN {X 0,Y 559.12,Z 140.333,A -85,B 0,C 180,E1 -2919.937,E2 -2919.937} C_VEL
LIN {X 0,Y 559.11,Z 140.342,A -85,B 0,C 180,E1 -2922.749,E2 -2922.749} C_VEL
LIN {X 0,Y 559.113,Z 140.334,A -85,B 0,C 180,E1 -2925.765,E2 -2925.765} C_VEL
LIN {X 0,Y 559.095,Z 140.339,A -85,B 0,C 180,E1 -2928.223,E2 -2928.223} C_VEL
LIN {X 0,Y 559.106,Z 140.339,A -85,B 0,C 180,E1 -2931.06,E2 -2931.06} C_VEL
LIN {X 0,Y 559.107,Z 140.335,A -85,B 0,C 180,E1 -2933.787,E2 -2933.787} C_VEL
LIN {X 0,Y 559.1,Z 140.343,A -85,B 0,C 180,E1 -2936.42,E2 -2936.42} C_VEL
LIN {X 0,Y 559.135,Z 140.335,A -85,B 0,C 180,E1 -2938.979,E2 -2938.979} C_VEL
LIN {X 0,Y 559.099,Z 140.337,A -85,B 0,C 180,E1 -2941.633,E2 -2941.633} C_VEL
LIN {X 0,Y 559.146,Z 140.333,A -85,B 0,C 180,E1 -2943.901,E2 -2943.901} C_VEL
LIN {X 0,Y 559.132,Z 140.426,A -85,B 0,C 180,E1 -2947.262,E2 -2947.262} C_VEL
LIN {X 0,Y 559.985,Z 146.156,A -85,B 0,C 180,E1 -2948.238,E2 -2948.238} C_VEL
LIN {X 0,Y 559.702,Z 163.442,A -85,B 0,C 180,E1 -2950.945,E2 -2950.945} C_VEL
LIN {X 0,Y 559.5,Z 179.293,A -85,B 0,C 180,E1 -2953.395,E2 -2953.395} C_VEL
LIN {X 0,Y 559.367,Z 195.206,A -85,B 0,C 180,E1 -2955.794,E2 -2955.794} C_VEL
LIN {X 0,Y 560.264,Z 202.159,A -85,B 0,C 180,E1 -2955.933,E2 -2955.933} C_VEL
LIN {X 0,Y 560.076,Z 302.917,A -85,B 0,C 180,E1 -2957.245,E2 -2957.245} C_VEL
LIN {X 0,Y 559.94,Z 316.197,A -85,B 0,C 180,E1 -2957.564,E2 -2957.564} C_VEL
LIN {X 0,Y 559.775,Z 328.362,A -85,B 0,C 180,E1 -2957.998,E2 -2957.998} C_VEL
LIN {X 0,Y 559.67,Z 339.802,A -85,B 0,C 180,E1 -2958.547,E2 -2958.547} C_VEL
LIN {X 0,Y 559.511,Z 350.893,A -85,B 0,C 180,E1 -2959.231,E2 -2959.231} C_VEL
LIN {X 0,Y 559.318,Z 361.529,A -85,B 0,C 180,E1 -2960.05,E2 -2960.05} C_VEL
LIN {X 0,Y 559.162,Z 371.107,A -85,B 0,C 180,E1 -2960.96,E2 -2960.96} C_VEL
LIN {X 0,Y 559.05,Z 378.955,A -85,B 0,C 180,E1 -2961.869,E2 -2961.869} C_VEL
LIN {X 0,Y 558.945,Z 386.619,A -85,B 0,C 180,E1 -2962.958,E2 -2962.958} C_VEL
LIN {X 0,Y 558.936,Z 393.676,A -85,B 0,C 180,E1 -2964.226,E2 -2964.226} C_VEL
LIN {X 0,Y 558.827,Z 398.37,A -85,B 0,C 180,E1 -2965.31,E2 -2965.31} C_VEL
LIN {X 0,Y 558.836,Z 401.956,A -85,B 0,C 180,E1 -2966.394,E2 -2966.394} C_VEL
LIN {X 0,Y 558.799,Z 403.805,A -85,B 0,C 180,E1 -2967.116,E2 -2967.116} C_VEL
LIN {X 0,Y 558.745,Z 406.182,A -85,B 0,C 180,E1 -2968.558,E2 -2968.558} C_VEL
LIN {X 0,Y 558.74,Z 407,A -85,B 0,C 180,E1 -2969.999,E2 -2969.999} C_VEL
LIN {X 0,Y 558.745,Z 406.185,A -85,B 0,C 180,E1 -2971.441,E2 -2971.441} C_VEL
LIN {X 0,Y 558.799,Z 403.812,A -85,B 0,C 180,E1 -2972.883,E2 -2972.883} C_VEL
LIN {X 0,Y 558.844,Z 400.898,A -85,B 0,C 180,E1 -2973.965,E2 -2973.965} C_VEL
LIN {X 0,Y 558.798,Z 396.951,A -85,B 0,C 180,E1 -2975.05,E2 -2975.05} C_VEL
LIN {X 0,Y 558.92,Z 391.872,A -85,B 0,C 180,E1 -2976.135,E2 -2976.135} C_VEL
LIN {X 0,Y 558.976,Z 385.473,A -85,B 0,C 180,E1 -2977.222,E2 -2977.222} C_VEL
LIN {X 0,Y 559.098,Z 377.484,A -85,B 0,C 180,E1 -2978.311,E2 -2978.311} C_VEL
LIN {X 0,Y 559.194,Z 369.342,A -85,B 0,C 180,E1 -2979.22,E2 -2979.22} C_VEL
LIN {X 0,Y 559.362,Z 359.408,A -85,B 0,C 180,E1 -2980.13,E2 -2980.13} C_VEL
LIN {X 0,Y 559.558,Z 348.376,A -85,B 0,C 180,E1 -2980.938,E2 -2980.938} C_VEL
LIN {X 0,Y 559.702,Z 336.155,A -85,B 0,C 180,E1 -2981.643,E2 -2981.643} C_VEL
LIN {X 0,Y 559.828,Z 323.795,A -85,B 0,C 180,E1 -2982.183,E2 -2982.183} C_VEL
LIN {X 0,Y 560.011,Z 310.382,A -85,B 0,C 180,E1 -2982.594,E2 -2982.594} C_VEL
LIN {X 0,Y 560.063,Z 297.143,A -85,B 0,C 180,E1 -2982.846,E2 -2982.846} C_VEL
LIN {X 0,Y 560.18,Z 200.812,A -85,B 0,C 180,E1 -2984.086,E2 -2984.086} C_VEL
LIN {X 0,Y 559.37,Z 195.204,A -85,B 0,C 180,E1 -2984.204,E2 -2984.204} C_VEL
LIN {X 0,Y 559.522,Z 176.196,A -85,B 0,C 180,E1 -2987.067,E2 -2987.067} C_VEL
LIN {X 0,Y 559.746,Z 159.364,A -85,B 0,C 180,E1 -2989.664,E2 -2989.664} C_VEL
LIN {X 0,Y 559.935,Z 145.172,A -85,B 0,C 180,E1 -2991.881,E2 -2991.881} C_VEL
LIN {X 0,Y 559.15,Z 140.461,A -85,B 0,C 180,E1 -2992.687,E2 -2992.687} C_VEL
LIN {X 0,Y 559.124,Z 140.34,A -85,B 0,C 180,E1 -2995.299,E2 -2995.299} C_VEL
LIN {X 0,Y 559.094,Z 140.345,A -85,B 0,C 180,E1 -2997.716,E2 -2997.716} C_VEL
LIN {X 0,Y 559.089,Z 140.34,A -85,B 0,C 180,E1 -3000.185,E2 -3000.185} C_VEL
LIN {X 0,Y 559.141,Z 140.332,A -85,B 0,C 180,E1 -3002.715,E2 -3002.715} C_VEL
LIN {X 0,Y 559.108,Z 140.343,A -85,B 0,C 180,E1 -3005.324,E2 -3005.324} C_VEL
LIN {X 0,Y 559.091,Z 140.339,A -85,B 0,C 180,E1 -3008.019,E2 -3008.019} C_VEL
LIN {X 0,Y 559.138,Z 140.333,A -85,B 0,C 180,E1 -3009.938,E2 -3009.938} C_VEL
LIN {X 0,Y 559.103,Z 140.337,A -85,B 0,C 180,E1 -3012.747,E2 -3012.747} C_VEL
LIN {X 0,Y 559.111,Z 140.337,A -85,B 0,C 180,E1 -3015.763,E2 -3015.763} C_VEL
LIN {X 0,Y 559.09,Z 140.337,A -85,B 0,C 180,E1 -3018.223,E2 -3018.223} C_VEL
LIN {X 0,Y 559.157,Z 140.336,A -85,B 0,C 180,E1 -3021.064,E2 -3021.064} C_VEL
LIN {X 0,Y 559.106,Z 140.337,A -85,B 0,C 180,E1 -3023.786,E2 -3023.786} C_VEL
LIN {X 0,Y 559.125,Z 140.333,A -85,B 0,C 180,E1 -3026.422,E2 -3026.422} C_VEL
LIN {X 0,Y 559.13,Z 140.34,A -85,B 0,C 180,E1 -3028.979,E2 -3028.979} C_VEL
LIN {X 0,Y 559.098,Z 140.337,A -85,B 0,C 180,E1 -3031.629,E2 -3031.629} C_VEL
LIN {X 0,Y 559.137,Z 140.331,A -85,B 0,C 180,E1 -3033.9,E2 -3033.9} C_VEL
LIN {X 0,Y 559.097,Z 140.344,A -85,B 0,C 180,E1 -3037.065,E2 -3037.065} C_VEL
LIN {X 0,Y 559.157,Z 140.331,A -85,B 0,C 180,E1 -3039.394,E2 -3039.394} C_VEL
LIN {X 0,Y 559.11,Z 140.334,A -85,B 0,C 180,E1 -3041.684,E2 -3041.684} C_VEL
LIN {X 0,Y 559.128,Z 140.332,A -85,B 0,C 180,E1 -3043.946,E2 -3043.946} C_VEL
LIN {X 0,Y 559.129,Z 140.333,A -85,B 0,C 180,E1 -3046.183,E2 -3046.183} C_VEL
LIN {X 0,Y 559.163,Z 140.331,A -85,B 0,C 180,E1 -3049.133,E2 -3049.133} C_VEL
LIN {X 0,Y 559.171,Z 140.328,A -85,B 0,C 180,E1 -3052.053,E2 -3052.053} C_VEL
LIN {X 0,Y 559.22,Z 140.325,A -85,B 0,C 180,E1 -3054.953,E2 -3054.953} C_VEL
LIN {X 0,Y 559.217,Z 140.322,A -85,B 0,C 180,E1 -3057.839,E2 -3057.839} C_VEL
LIN {X 0,Y 559.256,Z 140.324,A -85,B 0,C 180,E1 -3060.72,E2 -3060.72} C_VEL
LIN {X 0,Y 559.209,Z 140.325,A -85,B 0,C 180,E1 -3062.881,E2 -3062.881} C_VEL
LIN {X 0,Y 559.189,Z 140.326,A -85,B 0,C 180,E1 -3065.77,E2 -3065.77} C_VEL
LIN {X 0,Y 559.141,Z 140.336,A -85,B 0,C 180,E1 -3068.675,E2 -3068.675} C_VEL
LIN {X 0,Y 559.144,Z 140.331,A -85,B 0,C 180,E1 -3071.601,E2 -3071.601} C_VEL
LIN {X 0,Y 559.166,Z 140.333,A -85,B 0,C 180,E1 -3074.588,E2 -3074.588} C_VEL
LIN {X 0,Y 559.105,Z 140.336,A -85,B 0,C 180,E1 -3077.558,E2 -3077.558} C_VEL
LIN {X 0,Y 559.147,Z 140.334,A -85,B 0,C 180,E1 -3079.838,E2 -3079.838} C_VEL
LIN {X 0,Y 559.122,Z 140.343,A -85,B 0,C 180,E1 -3082.153,E2 -3082.153} C_VEL
LIN {X 0,Y 559.123,Z 140.333,A -85,B 0,C 180,E1 -3085.178,E2 -3085.178} C_VEL
LIN {X 0,Y 559.09,Z 140.342,A -85,B 0,C 180,E1 -3087.717,E2 -3087.717} C_VEL
LIN {X 0,Y 559.11,Z 140.338,A -85,B 0,C 180,E1 -3090.624,E2 -3090.624} C_VEL
LIN {X 0,Y 558.444,Z 140.421,A -85,B 0,C 180,E1 -3091.025,E2 -3091.025} C_VEL
LIN {X 0,Y 555.608,Z 140.777,A -85,B 0,C 180,E1 -3091.652,E2 -3091.652} C_VEL
LIN {X 0,Y 552.764,Z 141.134,A -85,B 0,C 180,E1 -3092.286,E2 -3092.286} C_VEL
LIN {X 0,Y 552.099,Z 141.213,A -85,B 0,C 180,E1 -3092.694,E2 -3092.694} C_VEL
LIN {X 0,Y 552.149,Z 141.423,A -85,B 0,C 180,E1 -3093.238,E2 -3093.238} C_VEL
LIN {X 0,Y 552.646,Z 145.82,A -85,B 0,C 180,E1 -3094.024,E2 -3094.024} C_VEL
LIN {X 0,Y 552.443,Z 162.945,A -85,B 0,C 180,E1 -3096.948,E2 -3096.948} C_VEL
LIN {X 0,Y 552.289,Z 179.13,A -85,B 0,C 180,E1 -3099.661,E2 -3099.661} C_VEL
LIN {X 0,Y 553.412,Z 186.446,A -85,B 0,C 180,E1 -3099.816,E2 -3099.816} C_VEL
LIN {X 0,Y 553.131,Z 286.539,A -85,B 0,C 180,E1 -3101.141,E2 -3101.141} C_VEL
LIN {X 0,Y 552.99,Z 299.188,A -85,B 0,C 180,E1 -3101.454,E2 -3101.454} C_VEL
LIN {X 0,Y 552.861,Z 309.452,A -85,B 0,C 180,E1 -3101.816,E2 -3101.816} C_VEL
LIN {X 0,Y 552.708,Z 319.865,A -85,B 0,C 180,E1 -3102.294,E2 -3102.294} C_VEL
LIN {X 0,Y 552.603,Z 328.311,A -85,B 0,C 180,E1 -3102.774,E2 -3102.774} C_VEL
LIN {X 0,Y 552.385,Z 337.424,A -85,B 0,C 180,E1 -3103.396,E2 -3103.396} C_VEL
LIN {X 0,Y 552.254,Z 346.233,A -85,B 0,C 180,E1 -3104.122,E2 -3104.122} C_VEL
LIN {X 0,Y 552.092,Z 354.277,A -85,B 0,C 180,E1 -3104.913,E2 -3104.913} C_VEL
LIN {X 0,Y 551.964,Z 361.877,A -85,B 0,C 180,E1 -3105.806,E2 -3105.806} C_VEL
LIN {X 0,Y 551.867,Z 370.477,A -85,B 0,C 180,E1 -3107.055,E2 -3107.055} C_VEL
LIN {X 0,Y 551.821,Z 376.035,A -85,B 0,C 180,E1 -3108.073,E2 -3108.073} C_VEL
LIN {X 0,Y 551.747,Z 380.577,A -85,B 0,C 180,E1 -3109.102,E2 -3109.102} C_VEL
LIN {X 0,Y 551.706,Z 383.319,A -85,B 0,C 180,E1 -3109.846,E2 -3109.846} C_VEL
LIN {X 0,Y 551.653,Z 386.498,A -85,B 0,C 180,E1 -3110.998,E2 -3110.998} C_VEL
LIN {X 0,Y 551.631,Z 388.796,A -85,B 0,C 180,E1 -3112.301,E2 -3112.301} C_VEL
LIN {X 0,Y 551.639,Z 389.762,A -85,B 0,C 180,E1 -3113.382,E2 -3113.382} C_VEL
LIN {X 0,Y 551.628,Z 389.989,A -85,B 0,C 180,E1 -3114.124,E2 -3114.124} C_VEL
LIN {X 0,Y 551.65,Z 389.634,A -85,B 0,C 180,E1 -3115.021,E2 -3115.021} C_VEL
LIN {X 0,Y 551.665,Z 388.651,A -85,B 0,C 180,E1 -3115.908,E2 -3115.908} C_VEL
LIN {X 0,Y 551.682,Z 386.212,A -85,B 0,C 180,E1 -3117.223,E2 -3117.223} C_VEL
LIN {X 0,Y 551.744,Z 382.08,A -85,B 0,C 180,E1 -3118.586,E2 -3118.586} C_VEL
LIN {X 0,Y 551.761,Z 377.441,A -85,B 0,C 180,E1 -3119.717,E2 -3119.717} C_VEL
LIN {X 0,Y 551.852,Z 372.721,A -85,B 0,C 180,E1 -3120.64,E2 -3120.64} C_VEL
LIN {X 0,Y 551.936,Z 366.191,A -85,B 0,C 180,E1 -3121.689,E2 -3121.689} C_VEL
LIN {X 0,Y 552.03,Z 359.993,A -85,B 0,C 180,E1 -3122.517,E2 -3122.517} C_VEL
LIN {X 0,Y 552.13,Z 353.957,A -85,B 0,C 180,E1 -3123.21,E2 -3123.21} C_VEL
LIN {X 0,Y 552.241,Z 346.352,A -85,B 0,C 180,E1 -3123.957,E2 -3123.957} C_VEL
LIN {X 0,Y 552.395,Z 338.704,A -85,B 0,C 180,E1 -3124.597,E2 -3124.597} C_VEL
LIN {X 0,Y 552.529,Z 330.442,A -85,B 0,C 180,E1 -3125.182,E2 -3125.182} C_VEL
LIN {X 0,Y 552.69,Z 319.971,A -85,B 0,C 180,E1 -3125.791,E2 -3125.791} C_VEL
LIN {X 0,Y 552.84,Z 310.095,A -85,B 0,C 180,E1 -3126.248,E2 -3126.248} C_VEL
LIN {X 0,Y 552.992,Z 299.572,A -85,B 0,C 180,E1 -3126.624,E2 -3126.624} C_VEL
LIN {X 0,Y 553.089,Z 287.793,A -85,B 0,C 180,E1 -3126.927,E2 -3126.927} C_VEL
LIN {X 0,Y 553.195,Z 251.651,A -85,B 0,C 180,E1 -3127.425,E2 -3127.425} C_VEL
LIN {X 0,Y 553.351,Z 186.108,A -85,B 0,C 180,E1 -3128.281,E2 -3128.281} C_VEL
LIN {X 0,Y 552.299,Z 179.434,A -85,B 0,C 180,E1 -3128.412,E2 -3128.412} C_VEL
LIN {X 0,Y 552.223,Z 178.306,A -85,B 0,C 180,E1 -3128.539,E2 -3128.539} C_VEL
LIN {X 0,Y 552.473,Z 162.512,A -85,B 0,C 180,E1 -3131.265,E2 -3131.265} C_VEL
LIN {X 0,Y 552.77,Z 146.082,A -85,B 0,C 180,E1 -3134.137,E2 -3134.137} C_VEL
LIN {X 0,Y 552.169,Z 141.244,A -85,B 0,C 180,E1 -3135.065,E2 -3135.065} C_VEL
LIN {X 0,Y 552.159,Z 141.208,A -85,B 0,C 180,E1 -3138.25,E2 -3138.25} C_VEL
LIN {X 0,Y 552.159,Z 141.202,A -85,B 0,C 180,E1 -3141.215,E2 -3141.215} C_VEL
LIN {X 0,Y 552.194,Z 141.201,A -85,B 0,C 180,E1 -3144.157,E2 -3144.157} C_VEL
LIN {X 0,Y 552.203,Z 141.195,A -85,B 0,C 180,E1 -3147.083,E2 -3147.083} C_VEL
LIN {X 0,Y 552.227,Z 141.197,A -85,B 0,C 180,E1 -3150.001,E2 -3150.001} C_VEL
LIN {X 0,Y 552.202,Z 141.195,A -85,B 0,C 180,E1 -3152.919,E2 -3152.919} C_VEL
LIN {X 0,Y 552.194,Z 141.202,A -85,B 0,C 180,E1 -3155.845,E2 -3155.845} C_VEL
LIN {X 0,Y 552.143,Z 141.203,A -85,B 0,C 180,E1 -3158.787,E2 -3158.787} C_VEL
LIN {X 0,Y 552.161,Z 141.205,A -85,B 0,C 180,E1 -3161.751,E2 -3161.751} C_VEL
LIN {X 0,Y 552.135,Z 141.204,A -85,B 0,C 180,E1 -3164.749,E2 -3164.749} C_VEL
LIN {X 0,Y 552.098,Z 141.211,A -85,B 0,C 180,E1 -3167.789,E2 -3167.789} C_VEL
LIN {X 0,Y 552.125,Z 141.205,A -85,B 0,C 180,E1 -3170.102,E2 -3170.102} C_VEL
LIN {X 0,Y 552.091,Z 141.209,A -85,B 0,C 180,E1 -3172.451,E2 -3172.451} C_VEL
LIN {X 0,Y 552.136,Z 141.21,A -85,B 0,C 180,E1 -3175.347,E2 -3175.347} C_VEL
LIN {X 0,Y 552.095,Z 141.208,A -85,B 0,C 180,E1 -3178.099,E2 -3178.099} C_VEL
LIN {X 0,Y 552.097,Z 141.211,A -85,B 0,C 180,E1 -3180.61,E2 -3180.61} C_VEL
LIN {X 0,Y 552.106,Z 141.214,A -85,B 0,C 180,E1 -3183.187,E2 -3183.187} C_VEL
LIN {X 0,Y 552.084,Z 141.21,A -85,B 0,C 180,E1 -3185.844,E2 -3185.844} C_VEL
LIN {X 0,Y 552.115,Z 141.21,A -85,B 0,C 180,E1 -3188.589,E2 -3188.589} C_VEL
LIN {X 0,Y 552.119,Z 141.207,A -85,B 0,C 180,E1 -3191.446,E2 -3191.446} C_VEL
LIN {X 0,Y 552.09,Z 141.215,A -85,B 0,C 180,E1 -3194.532,E2 -3194.532} C_VEL
LIN {X 0,Y 552.108,Z 141.207,A -85,B 0,C 180,E1 -3197.587,E2 -3197.587} C_VEL
LIN {X 0,Y 552.127,Z 141.211,A -85,B 0,C 180,E1 -3200.473,E2 -3200.473} C_VEL
LIN {X 0,Y 552.097,Z 141.209,A -85,B 0,C 180,E1 -3203.319,E2 -3203.319} C_VEL
LIN {X 0,Y 552.124,Z 141.206,A -85,B 0,C 180,E1 -3205.939,E2 -3205.939} C_VEL
LIN {X 0,Y 552.118,Z 141.214,A -85,B 0,C 180,E1 -3208.541,E2 -3208.541} C_VEL
LIN {X 0,Y 552.095,Z 141.208,A -85,B 0,C 180,E1 -3211.444,E2 -3211.444} C_VEL
LIN {X 0,Y 552.135,Z 141.208,A -85,B 0,C 180,E1 -3214.654,E2 -3214.654} C_VEL
LIN {X 0,Y 552.085,Z 141.21,A -85,B 0,C 180,E1 -3217.549,E2 -3217.549} C_VEL
LIN {X 0,Y 552.143,Z 141.209,A -85,B 0,C 180,E1 -3220.376,E2 -3220.376} C_VEL
LIN {X 0,Y 552.116,Z 141.206,A -85,B 0,C 180,E1 -3222.976,E2 -3222.976} C_VEL
LIN {X 0,Y 552.125,Z 141.213,A -85,B 0,C 180,E1 -3226.005,E2 -3226.005} C_VEL
LIN {X 0,Y 552.158,Z 141.2,A -85,B 0,C 180,E1 -3228.994,E2 -3228.994} C_VEL
LIN {X 0,Y 552.13,Z 141.214,A -85,B 0,C 180,E1 -3231.951,E2 -3231.951} C_VEL
LIN {X 0,Y 552.212,Z 141.194,A -85,B 0,C 180,E1 -3234.889,E2 -3234.889} C_VEL
LIN {X 0,Y 552.214,Z 141.203,A -85,B 0,C 180,E1 -3237.812,E2 -3237.812} C_VEL
LIN {X 0,Y 552.217,Z 141.199,A -85,B 0,C 180,E1 -3240,E2 -3240} C_VEL
LIN {X 0,Y 552.186,Z 141.197,A -85,B 0,C 180,E1 -3242.919,E2 -3242.919} C_VEL
LIN {X 0,Y 552.174,Z 141.205,A -85,B 0,C 180,E1 -3245.844,E2 -3245.844} C_VEL
LIN {X 0,Y 552.126,Z 141.205,A -85,B 0,C 180,E1 -3248.787,E2 -3248.787} C_VEL
LIN {X 0,Y 552.15,Z 141.207,A -85,B 0,C 180,E1 -3251.751,E2 -3251.751} C_VEL
LIN {X 0,Y 552.119,Z 141.206,A -85,B 0,C 180,E1 -3254.749,E2 -3254.749} C_VEL
LIN {X 0,Y 552.085,Z 141.213,A -85,B 0,C 180,E1 -3257.79,E2 -3257.79} C_VEL
LIN {X 0,Y 552.111,Z 141.207,A -85,B 0,C 180,E1 -3260.102,E2 -3260.102} C_VEL
LIN {X 0,Y 552.081,Z 141.21,A -85,B 0,C 180,E1 -3262.452,E2 -3262.452} C_VEL
LIN {X 0,Y 552.071,Z 141.219,A -85,B 0,C 180,E1 -3265.332,E2 -3265.332} C_VEL
LIN {X 0,Y 552.049,Z 141.214,A -85,B 0,C 180,E1 -3268.102,E2 -3268.102} C_VEL
LIN {X 0,Y 552.069,Z 141.214,A -85,B 0,C 180,E1 -3270.612,E2 -3270.612} C_VEL
LIN {X 0,Y 552.089,Z 141.217,A -85,B 0,C 180,E1 -3273.188,E2 -3273.188} C_VEL
LIN {X 0,Y 552.068,Z 141.212,A -85,B 0,C 180,E1 -3275.845,E2 -3275.845} C_VEL
LIN {X 0,Y 552.11,Z 141.21,A -85,B 0,C 180,E1 -3278.59,E2 -3278.59} C_VEL
LIN {X 0,Y 552.051,Z 141.215,A -85,B 0,C 180,E1 -3281.453,E2 -3281.453} C_VEL
LIN {X 0,Y 552.065,Z 141.217,A -85,B 0,C 180,E1 -3284.528,E2 -3284.528} C_VEL
LIN {X 0,Y 552.081,Z 141.21,A -85,B 0,C 180,E1 -3287.591,E2 -3287.591} C_VEL
LIN {X 0,Y 552.065,Z 141.218,A -85,B 0,C 180,E1 -3290.467,E2 -3290.467} C_VEL
LIN {X 0,Y 552.048,Z 141.215,A -85,B 0,C 180,E1 -3293.326,E2 -3293.326} C_VEL
LIN {X 0,Y 552.055,Z 141.215,A -85,B 0,C 180,E1 -3295.934,E2 -3295.934} C_VEL
LIN {X 0,Y 552.082,Z 141.219,A -85,B 0,C 180,E1 -3298.538,E2 -3298.538} C_VEL
LIN {X 0,Y 552.069,Z 141.213,A -85,B 0,C 180,E1 -3301.449,E2 -3301.449} C_VEL
LIN {X 0,Y 552.071,Z 141.221,A -85,B 0,C 180,E1 -3304.352,E2 -3304.352} C_VEL
LIN {X 0,Y 552.087,Z 141.294,A -85,B 0,C 180,E1 -3307.104,E2 -3307.104} C_VEL
LIN {X 0,Y 553.031,Z 146.864,A -85,B 0,C 180,E1 -3308.079,E2 -3308.079} C_VEL
LIN {X 0,Y 552.754,Z 161.75,A -85,B 0,C 180,E1 -3310.443,E2 -3310.443} C_VEL
LIN {X 0,Y 552.54,Z 177.98,A -85,B 0,C 180,E1 -3312.989,E2 -3312.989} C_VEL
LIN {X 0,Y 552.36,Z 195.129,A -85,B 0,C 180,E1 -3315.612,E2 -3315.612} C_VEL
LIN {X 0,Y 553.386,Z 202.714,A -85,B 0,C 180,E1 -3315.765,E2 -3315.765} C_VEL
LIN {X 0,Y 553.14,Z 302.667,A -85,B 0,C 180,E1 -3317.082,E2 -3317.082} C_VEL
LIN {X 0,Y 553.009,Z 316.011,A -85,B 0,C 180,E1 -3317.406,E2 -3317.406} C_VEL
LIN {X 0,Y 552.827,Z 328.208,A -85,B 0,C 180,E1 -3317.844,E2 -3317.844} C_VEL
LIN {X 0,Y 552.692,Z 340.544,A -85,B 0,C 180,E1 -3318.449,E2 -3318.449} C_VEL
LIN {X 0,Y 552.49,Z 352.11,A -85,B 0,C 180,E1 -3319.185,E2 -3319.185} C_VEL
LIN {X 0,Y 552.277,Z 362.552,A -85,B 0,C 180,E1 -3320.015,E2 -3320.015} C_VEL
LIN {X 0,Y 552.132,Z 371.087,A -85,B 0,C 180,E1 -3320.844,E2 -3320.844} C_VEL
LIN {X 0,Y 552.013,Z 378.955,A -85,B 0,C 180,E1 -3321.765,E2 -3321.765} C_VEL
LIN {X 0,Y 551.89,Z 386.617,A -85,B 0,C 180,E1 -3322.867,E2 -3322.867} C_VEL
LIN {X 0,Y 551.868,Z 393.676,A -85,B 0,C 180,E1 -3324.152,E2 -3324.152} C_VEL
LIN {X 0,Y 551.725,Z 398.37,A -85,B 0,C 180,E1 -3325.25,E2 -3325.25} C_VEL
LIN {X 0,Y 551.751,Z 401.956,A -85,B 0,C 180,E1 -3326.348,E2 -3326.348} C_VEL
LIN {X 0,Y 551.724,Z 403.805,A -85,B 0,C 180,E1 -3327.079,E2 -3327.079} C_VEL
LIN {X 0,Y 551.645,Z 406.181,A -85,B 0,C 180,E1 -3328.539,E2 -3328.539} C_VEL
LIN {X 0,Y 551.64,Z 407,A -85,B 0,C 180,E1 -3329.999,E2 -3329.999} C_VEL
LIN {X 0,Y 551.645,Z 406.184,A -85,B 0,C 180,E1 -3331.459,E2 -3331.459} C_VEL
LIN {X 0,Y 551.723,Z 403.812,A -85,B 0,C 180,E1 -3332.92,E2 -3332.92} C_VEL
LIN {X 0,Y 551.764,Z 400.898,A -85,B 0,C 180,E1 -3334.016,E2 -3334.016} C_VEL
LIN {X 0,Y 551.723,Z 396.951,A -85,B 0,C 180,E1 -3335.115,E2 -3335.115} C_VEL
LIN {X 0,Y 551.823,Z 391.199,A -85,B 0,C 180,E1 -3336.339,E2 -3336.339} C_VEL
LIN {X 0,Y 551.926,Z 384.241,A -85,B 0,C 180,E1 -3337.499,E2 -3337.499} C_VEL
LIN {X 0,Y 552.082,Z 375.994,A -85,B 0,C 180,E1 -3338.602,E2 -3338.602} C_VEL
LIN {X 0,Y 552.2,Z 367.517,A -85,B 0,C 180,E1 -3339.523,E2 -3339.523} C_VEL
LIN {X 0,Y 552.436,Z 357.039,A -85,B 0,C 180,E1 -3340.444,E2 -3340.444} C_VEL
LIN {X 0,Y 552.6,Z 346.044,A -85,B 0,C 180,E1 -3341.223,E2 -3341.223} C_VEL
LIN {X 0,Y 552.752,Z 335.291,A -85,B 0,C 180,E1 -3341.83,E2 -3341.83} C_VEL
LIN {X 0,Y 552.878,Z 323.612,A -85,B 0,C 180,E1 -3342.339,E2 -3342.339} C_VEL
LIN {X 0,Y 553.079,Z 310.148,A -85,B 0,C 180,E1 -3342.754,E2 -3342.754} C_VEL
LIN {X 0,Y 553.163,Z 296.807,A -85,B 0,C 180,E1 -3343.009,E2 -3343.009} C_VEL
LIN {X 0,Y 553.311,Z 201.69,A -85,B 0,C 180,E1 -3344.251,E2 -3344.251} C_VEL
LIN {X 0,Y 552.336,Z 195.092,A -85,B 0,C 180,E1 -3344.387,E2 -3344.387} C_VEL
LIN {X 0,Y 552.517,Z 176.771,A -85,B 0,C 180,E1 -3347.178,E2 -3347.178} C_VEL
LIN {X 0,Y 552.776,Z 159.95,A -85,B 0,C 180,E1 -3349.807,E2 -3349.807} C_VEL
LIN {X 0,Y 552.988,Z 146.646,A -85,B 0,C 180,E1 -3351.91,E2 -3351.91} C_VEL
LIN {X 0,Y 552.075,Z 141.295,A -85,B 0,C 180,E1 -3352.846,E2 -3352.846} C_VEL
LIN {X 0,Y 552.078,Z 141.22,A -85,B 0,C 180,E1 -3355.646,E2 -3355.646} C_VEL
LIN {X 0,Y 552.065,Z 141.214,A -85,B 0,C 180,E1 -3358.55,E2 -3358.55} C_VEL
LIN {X 0,Y 552.087,Z 141.218,A -85,B 0,C 180,E1 -3361.471,E2 -3361.471} C_VEL
LIN {X 0,Y 552.089,Z 141.211,A -85,B 0,C 180,E1 -3364.163,E2 -3364.163} C_VEL
LIN {X 0,Y 552.045,Z 141.216,A -85,B 0,C 180,E1 -3366.75,E2 -3366.75} C_VEL
LIN {X 0,Y 552.082,Z 141.218,A -85,B 0,C 180,E1 -3369.53,E2 -3369.53} C_VEL
LIN {X 0,Y 552.072,Z 141.212,A -85,B 0,C 180,E1 -3372.429,E2 -3372.429} C_VEL
LIN {X 0,Y 552.062,Z 141.218,A -85,B 0,C 180,E1 -3375.559,E2 -3375.559} C_VEL
LIN {X 0,Y 552.05,Z 141.215,A -85,B 0,C 180,E1 -3378.547,E2 -3378.547} C_VEL
LIN {X 0,Y 552.099,Z 141.213,A -85,B 0,C 180,E1 -3381.409,E2 -3381.409} C_VEL
LIN {X 0,Y 552.06,Z 141.213,A -85,B 0,C 180,E1 -3384.154,E2 -3384.154} C_VEL
LIN {X 0,Y 552.085,Z 141.219,A -85,B 0,C 180,E1 -3387.156,E2 -3387.156} C_VEL
LIN {X 0,Y 552.065,Z 141.212,A -85,B 0,C 180,E1 -3389.956,E2 -3389.956} C_VEL
LIN {X 0,Y 552.078,Z 141.218,A -85,B 0,C 180,E1 -3393.009,E2 -3393.009} C_VEL
LIN {X 0,Y 552.06,Z 141.212,A -85,B 0,C 180,E1 -3395.96,E2 -3395.96} C_VEL
LIN {X 0,Y 552.101,Z 141.213,A -85,B 0,C 180,E1 -3399.119,E2 -3399.119} C_VEL
LIN {X 0,Y 552.07,Z 141.213,A -85,B 0,C 180,E1 -3401.442,E2 -3401.442} C_VEL
LIN {X 0,Y 552.077,Z 141.21,A -85,B 0,C 180,E1 -3403.736,E2 -3403.736} C_VEL
LIN {X 0,Y 552.091,Z 141.209,A -85,B 0,C 180,E1 -3406.003,E2 -3406.003} C_VEL
LIN {X 0,Y 552.136,Z 141.209,A -85,B 0,C 180,E1 -3408.993,E2 -3408.993} C_VEL
LIN {X 0,Y 552.126,Z 141.205,A -85,B 0,C 180,E1 -3411.951,E2 -3411.951} C_VEL
LIN {X 0,Y 552.197,Z 141.201,A -85,B 0,C 180,E1 -3414.888,E2 -3414.888} C_VEL
LIN {X 0,Y 552.19,Z 141.197,A -85,B 0,C 180,E1 -3417.811,E2 -3417.811} C_VEL
LIN {X 0,Y 552.225,Z 141.199,A -85,B 0,C 180,E1 -3420.729,E2 -3420.729} C_VEL
LIN {X 0,Y 552.174,Z 141.201,A -85,B 0,C 180,E1 -3422.918,E2 -3422.918} C_VEL
LIN {X 0,Y 552.162,Z 141.202,A -85,B 0,C 180,E1 -3425.844,E2 -3425.844} C_VEL
LIN {X 0,Y 552.114,Z 141.21,A -85,B 0,C 180,E1 -3428.786,E2 -3428.786} C_VEL
LIN {X 0,Y 552.094,Z 141.21,A -85,B 0,C 180,E1 -3431.752,E2 -3431.752} C_VEL
LIN {X 0,Y 552.113,Z 141.21,A -85,B 0,C 180,E1 -3434.749,E2 -3434.749} C_VEL
LIN {X 0,Y 552.067,Z 141.215,A -85,B 0,C 180,E1 -3437.79,E2 -3437.79} C_VEL
LIN {X 0,Y 552.108,Z 141.215,A -85,B 0,C 180,E1 -3440.102,E2 -3440.102} C_VEL
LIN {X 0,Y 552.073,Z 141.217,A -85,B 0,C 180,E1 -3442.451,E2 -3442.451} C_VEL
LIN {X 0,Y 552.066,Z 141.212,A -85,B 0,C 180,E1 -3445.334,E2 -3445.334} C_VEL
LIN {X 0,Y 552.039,Z 141.224,A -85,B 0,C 180,E1 -3448.102,E2 -3448.102} C_VEL
LIN {X 0,Y 552.074,Z 141.216,A -85,B 0,C 180,E1 -3450.62,E2 -3450.62} C_VEL
LIN {X 0,Y 552.099,Z 141.213,A -85,B 0,C 180,E1 -3452.694,E2 -3452.694} C_VEL
LIN {X 0,Y 551.813,Z 141.795,A -85,B 0,C 180,E1 -3453.097,E2 -3453.097} C_VEL
LIN {X 0,Y 550.594,Z 144.188,A -85,B 0,C 180,E1 -3453.653,E2 -3453.653} C_VEL
LIN {X 0,Y 546.656,Z 151.772,A -85,B 0,C 180,E1 -3454.834,E2 -3454.834} C_VEL
LIN {X 0,Y 545.646,Z 154.986,A -85,B 0,C 180,E1 -3455.354,E2 -3455.354} C_VEL
LIN {X 0,Y 545.549,Z 156.038,A -85,B 0,C 180,E1 -3455.532,E2 -3455.532} C_VEL
LIN {X 0,Y 545.316,Z 173,A -85,B 0,C 180,E1 -3458.45,E2 -3458.45} C_VEL
LIN {X 0,Y 545.272,Z 179.159,A -85,B 0,C 180,E1 -3459.467,E2 -3459.467} C_VEL
LIN {X 0,Y 546.289,Z 185.195,A -85,B 0,C 180,E1 -3459.608,E2 -3459.608} C_VEL
LIN {X 0,Y 546.533,Z 192.006,A -85,B 0,C 180,E1 -3459.706,E2 -3459.706} C_VEL
LIN {X 0,Y 546.217,Z 286.878,A -85,B 0,C 180,E1 -3460.982,E2 -3460.982} C_VEL
LIN {X 0,Y 546.085,Z 299.356,A -85,B 0,C 180,E1 -3461.296,E2 -3461.296} C_VEL
LIN {X 0,Y 545.912,Z 310.467,A -85,B 0,C 180,E1 -3461.698,E2 -3461.698} C_VEL
LIN {X 0,Y 545.757,Z 320.324,A -85,B 0,C 180,E1 -3462.162,E2 -3462.162} C_VEL
LIN {X 0,Y 545.578,Z 330.437,A -85,B 0,C 180,E1 -3462.757,E2 -3462.757} C_VEL
LIN {X 0,Y 545.359,Z 341.748,A -85,B 0,C 180,E1 -3463.586,E2 -3463.586} C_VEL
LIN {X 0,Y 545.149,Z 351.143,A -85,B 0,C 180,E1 -3464.45,E2 -3464.45} C_VEL
LIN {X 0,Y 544.978,Z 359.188,A -85,B 0,C 180,E1 -3465.348,E2 -3465.348} C_VEL
LIN {X 0,Y 544.856,Z 365.939,A -85,B 0,C 180,E1 -3466.247,E2 -3466.247} C_VEL
LIN {X 0,Y 544.796,Z 371.525,A -85,B 0,C 180,E1 -3467.131,E2 -3467.131} C_VEL
LIN {X 0,Y 544.719,Z 376.99,A -85,B 0,C 180,E1 -3468.182,E2 -3468.182} C_VEL
LIN {X 0,Y 544.668,Z 381.417,A -85,B 0,C 180,E1 -3469.244,E2 -3469.244} C_VEL
LIN {X 0,Y 544.607,Z 384.838,A -85,B 0,C 180,E1 -3470.301,E2 -3470.301} C_VEL
LIN {X 0,Y 544.56,Z 386.155,A -85,B 0,C 180,E1 -3470.775,E2 -3470.775} C_VEL
LIN {X 0,Y 544.529,Z 388.435,A -85,B 0,C 180,E1 -3471.933,E2 -3471.933} C_VEL
LIN {X 0,Y 544.554,Z 389.724,A -85,B 0,C 180,E1 -3473.146,E2 -3473.146} C_VEL
LIN {X 0,Y 544.55,Z 389.898,A -85,B 0,C 180,E1 -3474.497,E2 -3474.497} C_VEL
LIN {X 0,Y 544.562,Z 388.995,A -85,B 0,C 180,E1 -3475.686,E2 -3475.686} C_VEL
LIN {X 0,Y 544.553,Z 388.21,A -85,B 0,C 180,E1 -3476.294,E2 -3476.294} C_VEL
LIN {X 0,Y 544.62,Z 385.304,A -85,B 0,C 180,E1 -3477.621,E2 -3477.621} C_VEL
LIN {X 0,Y 544.656,Z 383.086,A -85,B 0,C 180,E1 -3478.389,E2 -3478.389} C_VEL
LIN {X 0,Y 544.681,Z 379.487,A -85,B 0,C 180,E1 -3479.36,E2 -3479.36} C_VEL
LIN {X 0,Y 544.772,Z 373.274,A -85,B 0,C 180,E1 -3480.646,E2 -3480.646} C_VEL
LIN {X 0,Y 544.829,Z 368.276,A -85,B 0,C 180,E1 -3481.493,E2 -3481.493} C_VEL
LIN {X 0,Y 544.955,Z 361.249,A -85,B 0,C 180,E1 -3482.482,E2 -3482.482} C_VEL
LIN {X 0,Y 545.099,Z 353.539,A -85,B 0,C 180,E1 -3483.384,E2 -3483.384} C_VEL
LIN {X 0,Y 545.259,Z 345.884,A -85,B 0,C 180,E1 -3484.137,E2 -3484.137} C_VEL
LIN {X 0,Y 545.465,Z 336.071,A -85,B 0,C 180,E1 -3484.941,E2 -3484.941} C_VEL
LIN {X 0,Y 545.702,Z 324.096,A -85,B 0,C 180,E1 -3485.727,E2 -3485.727} C_VEL
LIN {X 0,Y 545.885,Z 312.577,A -85,B 0,C 180,E1 -3486.303,E2 -3486.303} C_VEL
LIN {X 0,Y 546.028,Z 301.18,A -85,B 0,C 180,E1 -3486.736,E2 -3486.736} C_VEL
LIN {X 0,Y 546.163,Z 288.939,A -85,B 0,C 180,E1 -3487.068,E2 -3487.068} C_VEL
LIN {X 0,Y 546.294,Z 266.335,A -85,B 0,C 180,E1 -3487.402,E2 -3487.402} C_VEL
LIN {X 0,Y 546.41,Z 186.1,A -85,B 0,C 180,E1 -3488.467,E2 -3488.467} C_VEL
LIN {X 0,Y 545.258,Z 179.392,A -85,B 0,C 180,E1 -3488.609,E2 -3488.609} C_VEL
LIN {X 0,Y 545.309,Z 174.297,A -85,B 0,C 180,E1 -3489.44,E2 -3489.44} C_VEL
LIN {X 0,Y 545.555,Z 157.343,A -85,B 0,C 180,E1 -3492.417,E2 -3492.417} C_VEL
LIN {X 0,Y 545.69,Z 145.62,A -85,B 0,C 180,E1 -3494.501,E2 -3494.501} C_VEL
LIN {X 0,Y 545.149,Z 142.133,A -85,B 0,C 180,E1 -3495.194,E2 -3495.194} C_VEL
LIN {X 0,Y 545.133,Z 142.081,A -85,B 0,C 180,E1 -3498.466,E2 -3498.466} C_VEL
LIN {X 0,Y 545.117,Z 142.078,A -85,B 0,C 180,E1 -3501.101,E2 -3501.101} C_VEL
LIN {X 0,Y 545.166,Z 142.078,A -85,B 0,C 180,E1 -3504.081,E2 -3504.081} C_VEL
LIN {X 0,Y 545.169,Z 142.071,A -85,B 0,C 180,E1 -3507.045,E2 -3507.045} C_VEL
LIN {X 0,Y 545.198,Z 142.073,A -85,B 0,C 180,E1 -3510.001,E2 -3510.001} C_VEL
LIN {X 0,Y 545.169,Z 142.072,A -85,B 0,C 180,E1 -3512.957,E2 -3512.957} C_VEL
LIN {X 0,Y 545.166,Z 142.076,A -85,B 0,C 180,E1 -3515.92,E2 -3515.92} C_VEL
LIN {X 0,Y 545.106,Z 142.08,A -85,B 0,C 180,E1 -3518.901,E2 -3518.901} C_VEL
LIN {X 0,Y 545.134,Z 142.079,A -85,B 0,C 180,E1 -3521.905,E2 -3521.905} C_VEL
LIN {X 0,Y 545.084,Z 142.084,A -85,B 0,C 180,E1 -3524.944,E2 -3524.944} C_VEL
LIN {X 0,Y 545.069,Z 142.084,A -85,B 0,C 180,E1 -3528.027,E2 -3528.027} C_VEL
LIN {X 0,Y 545.091,Z 142.081,A -85,B 0,C 180,E1 -3530.373,E2 -3530.373} C_VEL
LIN {X 0,Y 545.079,Z 142.087,A -85,B 0,C 180,E1 -3533.56,E2 -3533.56} C_VEL
LIN {X 0,Y 545.077,Z 142.083,A -85,B 0,C 180,E1 -3536.001,E2 -3536.001} C_VEL
LIN {X 0,Y 545.073,Z 142.087,A -85,B 0,C 180,E1 -3538.746,E2 -3538.746} C_VEL
LIN {X 0,Y 545.057,Z 142.086,A -85,B 0,C 180,E1 -3541.679,E2 -3541.679} C_VEL
LIN {X 0,Y 545.058,Z 142.088,A -85,B 0,C 180,E1 -3544.565,E2 -3544.565} C_VEL
LIN {X 0,Y 545.034,Z 142.092,A -85,B 0,C 180,E1 -3547.304,E2 -3547.304} C_VEL
LIN {X 0,Y 545.063,Z 142.085,A -85,B 0,C 180,E1 -3550.143,E2 -3550.143} C_VEL
LIN {X 0,Y 545.077,Z 142.087,A -85,B 0,C 180,E1 -3553.107,E2 -3553.107} C_VEL
LIN {X 0,Y 545.048,Z 142.088,A -85,B 0,C 180,E1 -3556.227,E2 -3556.227} C_VEL
LIN {X 0,Y 545.079,Z 142.088,A -85,B 0,C 180,E1 -3558.886,E2 -3558.886} C_VEL
LIN {X 0,Y 545.077,Z 142.089,A -85,B 0,C 180,E1 -3560.818,E2 -3560.818} C_VEL
LIN {X 0,Y 545.032,Z 142.088,A -85,B 0,C 180,E1 -3563.619,E2 -3563.619} C_VEL
LIN {X 0,Y 545.063,Z 142.091,A -85,B 0,C 180,E1 -3566.328,E2 -3566.328} C_VEL
LIN {X 0,Y 545.064,Z 142.087,A -85,B 0,C 180,E1 -3568.952,E2 -3568.952} C_VEL
LIN {X 0,Y 545.073,Z 142.083,A -85,B 0,C 180,E1 -3571.506,E2 -3571.506} C_VEL
LIN {X 0,Y 545.103,Z 142.082,A -85,B 0,C 180,E1 -3574.82,E2 -3574.82} C_VEL
LIN {X 0,Y 545.03,Z 142.088,A -85,B 0,C 180,E1 -3577.242,E2 -3577.242} C_VEL
LIN {X 0,Y 545.114,Z 142.084,A -85,B 0,C 180,E1 -3580.415,E2 -3580.415} C_VEL
LIN {X 0,Y 545.043,Z 142.088,A -85,B 0,C 180,E1 -3583.521,E2 -3583.521} C_VEL
LIN {X 0,Y 545.08,Z 142.087,A -85,B 0,C 180,E1 -3585.82,E2 -3585.82} C_VEL
LIN {X 0,Y 545.115,Z 142.078,A -85,B 0,C 180,E1 -3588.85,E2 -3588.85} C_VEL
LIN {X 0,Y 545.082,Z 142.09,A -85,B 0,C 180,E1 -3591.847,E2 -3591.847} C_VEL
LIN {X 0,Y 545.169,Z 142.071,A -85,B 0,C 180,E1 -3594.823,E2 -3594.823} C_VEL
LIN {X 0,Y 545.186,Z 142.078,A -85,B 0,C 180,E1 -3597.784,E2 -3597.784} C_VEL
LIN {X 0,Y 545.186,Z 142.075,A -85,B 0,C 180,E1 -3600,E2 -3600} C_VEL
LIN {X 0,Y 545.155,Z 142.073,A -85,B 0,C 180,E1 -3602.956,E2 -3602.956} C_VEL
LIN {X 0,Y 545.121,Z 142.082,A -85,B 0,C 180,E1 -3605.92,E2 -3605.92} C_VEL
LIN {X 0,Y 545.07,Z 142.084,A -85,B 0,C 180,E1 -3608.901,E2 -3608.901} C_VEL
LIN {X 0,Y 545.093,Z 142.084,A -85,B 0,C 180,E1 -3611.905,E2 -3611.905} C_VEL
LIN {X 0,Y 545.075,Z 142.085,A -85,B 0,C 180,E1 -3614.944,E2 -3614.944} C_VEL
LIN {X 0,Y 545.052,Z 142.087,A -85,B 0,C 180,E1 -3618.027,E2 -3618.027} C_VEL
LIN {X 0,Y 545.049,Z 142.086,A -85,B 0,C 180,E1 -3620.374,E2 -3620.374} C_VEL
LIN {X 0,Y 545.026,Z 142.091,A -85,B 0,C 180,E1 -3622.759,E2 -3622.759} C_VEL
LIN {X 0,Y 545.022,Z 142.095,A -85,B 0,C 180,E1 -3625.493,E2 -3625.493} C_VEL
LIN {X 0,Y 545.033,Z 142.089,A -85,B 0,C 180,E1 -3628.497,E2 -3628.497} C_VEL
LIN {X 0,Y 545.043,Z 142.088,A -85,B 0,C 180,E1 -3631.676,E2 -3631.676} C_VEL
LIN {X 0,Y 545.043,Z 142.089,A -85,B 0,C 180,E1 -3634.566,E2 -3634.566} C_VEL
LIN {X 0,Y 545.012,Z 142.095,A -85,B 0,C 180,E1 -3637.306,E2 -3637.306} C_VEL
LIN {X 0,Y 545.05,Z 142.089,A -85,B 0,C 180,E1 -3639.317,E2 -3639.317} C_VEL
LIN {X 0,Y 545.029,Z 142.089,A -85,B 0,C 180,E1 -3642.108,E2 -3642.108} C_VEL
LIN {X 0,Y 545.013,Z 142.094,A -85,B 0,C 180,E1 -3645.173,E2 -3645.173} C_VEL
LIN {X 0,Y 545.022,Z 142.094,A -85,B 0,C 180,E1 -3648.41,E2 -3648.41} C_VEL
LIN {X 0,Y 545.023,Z 142.097,A -85,B 0,C 180,E1 -3650.813,E2 -3650.813} C_VEL
LIN {X 0,Y 544.996,Z 142.092,A -85,B 0,C 180,E1 -3653.616,E2 -3653.616} C_VEL
LIN {X 0,Y 545.041,Z 142.09,A -85,B 0,C 180,E1 -3656.945,E2 -3656.945} C_VEL
LIN {X 0,Y 545.018,Z 142.092,A -85,B 0,C 180,E1 -3659.807,E2 -3659.807} C_VEL
LIN {X 0,Y 545.022,Z 142.093,A -85,B 0,C 180,E1 -3662.842,E2 -3662.842} C_VEL
LIN {X 0,Y 545.009,Z 142.096,A -85,B 0,C 180,E1 -3665.628,E2 -3665.628} C_VEL
LIN {X 0,Y 545.079,Z 142.308,A -85,B 0,C 180,E1 -3666.993,E2 -3666.993} C_VEL
LIN {X 0,Y 546.06,Z 148.614,A -85,B 0,C 180,E1 -3668.084,E2 -3668.084} C_VEL
LIN {X 0,Y 545.806,Z 161.506,A -85,B 0,C 180,E1 -3670.16,E2 -3670.16} C_VEL
LIN {X 0,Y 545.562,Z 177.886,A -85,B 0,C 180,E1 -3672.765,E2 -3672.765} C_VEL
LIN {X 0,Y 545.342,Z 194.994,A -85,B 0,C 180,E1 -3675.422,E2 -3675.422} C_VEL
LIN {X 0,Y 546.516,Z 203.543,A -85,B 0,C 180,E1 -3675.595,E2 -3675.595} C_VEL
LIN {X 0,Y 546.233,Z 302.413,A -85,B 0,C 180,E1 -3676.916,E2 -3676.916} C_VEL
LIN {X 0,Y 546.066,Z 315.808,A -85,B 0,C 180,E1 -3677.243,E2 -3677.243} C_VEL
LIN {X 0,Y 545.865,Z 328.028,A -85,B 0,C 180,E1 -3677.687,E2 -3677.687} C_VEL
LIN {X 0,Y 545.686,Z 340.385,A -85,B 0,C 180,E1 -3678.298,E2 -3678.298} C_VEL
LIN {X 0,Y 545.499,Z 351.961,A -85,B 0,C 180,E1 -3679.045,E2 -3679.045} C_VEL
LIN {X 0,Y 545.265,Z 362.411,A -85,B 0,C 180,E1 -3679.885,E2 -3679.885} C_VEL
LIN {X 0,Y 545.088,Z 370.952,A -85,B 0,C 180,E1 -3680.725,E2 -3680.725} C_VEL
LIN {X 0,Y 544.945,Z 378.829,A -85,B 0,C 180,E1 -3681.657,E2 -3681.657} C_VEL
LIN {X 0,Y 544.825,Z 386.519,A -85,B 0,C 180,E1 -3682.774,E2 -3682.774} C_VEL
LIN {X 0,Y 544.777,Z 393.604,A -85,B 0,C 180,E1 -3684.076,E2 -3684.076} C_VEL
LIN {X 0,Y 544.629,Z 398.314,A -85,B 0,C 180,E1 -3685.188,E2 -3685.188} C_VEL
LIN {X 0,Y 544.669,Z 401.914,A -85,B 0,C 180,E1 -3686.3,E2 -3686.3} C_VEL
LIN {X 0,Y 544.651,Z 403.77,A -85,B 0,C 180,E1 -3687.041,E2 -3687.041} C_VEL
LIN {X 0,Y 544.546,Z 406.153,A -85,B 0,C 180,E1 -3688.52,E2 -3688.52} C_VEL
LIN {X 0,Y 544.541,Z 406.975,A -85,B 0,C 180,E1 -3689.999,E2 -3689.999} C_VEL
LIN {X 0,Y 544.546,Z 406.156,A -85,B 0,C 180,E1 -3691.478,E2 -3691.478} C_VEL
LIN {X 0,Y 544.65,Z 403.776,A -85,B 0,C 180,E1 -3692.958,E2 -3692.958} C_VEL
LIN {X 0,Y 544.684,Z 400.851,A -85,B 0,C 180,E1 -3694.069,E2 -3694.069} C_VEL
LIN {X 0,Y 544.653,Z 396.888,A -85,B 0,C 180,E1 -3695.181,E2 -3695.181} C_VEL
LIN {X 0,Y 544.732,Z 391.521,A -85,B 0,C 180,E1 -3696.347,E2 -3696.347} C_VEL
LIN {X 0,Y 544.859,Z 384.129,A -85,B 0,C 180,E1 -3697.597,E2 -3697.597} C_VEL
LIN {X 0,Y 545.007,Z 375.856,A -85,B 0,C 180,E1 -3698.714,E2 -3698.714} C_VEL
LIN {X 0,Y 545.154,Z 367.371,A -85,B 0,C 180,E1 -3699.647,E2 -3699.647} C_VEL
LIN {X 0,Y 545.407,Z 356.883,A -85,B 0,C 180,E1 -3700.58,E2 -3700.58} C_VEL
LIN {X 0,Y 545.615,Z 345.1,A -85,B 0,C 180,E1 -3701.42,E2 -3701.42} C_VEL
LIN {X 0,Y 545.827,Z 333.179,A -85,B 0,C 180,E1 -3702.076,E2 -3702.076} C_VEL
LIN {X 0,Y 546.002,Z 320.799,A -85,B 0,C 180,E1 -3702.591,E2 -3702.591} C_VEL
LIN {X 0,Y 546.164,Z 308.07,A -85,B 0,C 180,E1 -3702.966,E2 -3702.966} C_VEL
LIN {X 0,Y 546.272,Z 292.912,A -85,B 0,C 180,E1 -3703.223,E2 -3703.223} C_VEL
LIN {X 0,Y 546.435,Z 202.33,A -85,B 0,C 180,E1 -3704.423,E2 -3704.423} C_VEL
LIN {X 0,Y 545.345,Z 195.024,A -85,B 0,C 180,E1 -3704.573,E2 -3704.573} C_VEL
LIN {X 0,Y 545.556,Z 176.266,A -85,B 0,C 180,E1 -3707.463,E2 -3707.463} C_VEL
LIN {X 0,Y 545.91,Z 156.877,A -85,B 0,C 180,E1 -3710.536,E2 -3710.536} C_VEL
LIN {X 0,Y 545.989,Z 147.388,A -85,B 0,C 180,E1 -3712.06,E2 -3712.06} C_VEL
LIN {X 0,Y 545.051,Z 142.187,A -85,B 0,C 180,E1 -3712.981,E2 -3712.981} C_VEL
LIN {X 0,Y 545.037,Z 142.094,A -85,B 0,C 180,E1 -3716.001,E2 -3716.001} C_VEL
LIN {X 0,Y 545.011,Z 142.093,A -85,B 0,C 180,E1 -3718.732,E2 -3718.732} C_VEL
LIN {X 0,Y 545.04,Z 142.092,A -85,B 0,C 180,E1 -3721.914,E2 -3721.914} C_VEL
LIN {X 0,Y 545.039,Z 142.089,A -85,B 0,C 180,E1 -3724.565,E2 -3724.565} C_VEL
LIN {X 0,Y 544.996,Z 142.101,A -85,B 0,C 180,E1 -3727.306,E2 -3727.306} C_VEL
LIN {X 0,Y 545.039,Z 142.088,A -85,B 0,C 180,E1 -3730.143,E2 -3730.143} C_VEL
LIN {X 0,Y 544.99,Z 142.1,A -85,B 0,C 180,E1 -3733.113,E2 -3733.113} C_VEL
LIN {X 0,Y 545.02,Z 142.092,A -85,B 0,C 180,E1 -3735.867,E2 -3735.867} C_VEL
LIN {X 0,Y 545.005,Z 142.096,A -85,B 0,C 180,E1 -3738.878,E2 -3738.878} C_VEL
LIN {X 0,Y 545.032,Z 142.089,A -85,B 0,C 180,E1 -3741.761,E2 -3741.761} C_VEL
LIN {X 0,Y 545.015,Z 142.092,A -85,B 0,C 180,E1 -3744.53,E2 -3744.53} C_VEL
LIN {X 0,Y 545.04,Z 142.095,A -85,B 0,C 180,E1 -3747.209,E2 -3747.209} C_VEL
LIN {X 0,Y 545.014,Z 142.091,A -85,B 0,C 180,E1 -3749.807,E2 -3749.807} C_VEL
LIN {X 0,Y 545.022,Z 142.096,A -85,B 0,C 180,E1 -3752.838,E2 -3752.838} C_VEL
LIN {X 0,Y 545.003,Z 142.092,A -85,B 0,C 180,E1 -3755.628,E2 -3755.628} C_VEL
LIN {X 0,Y 545.051,Z 142.086,A -85,B 0,C 180,E1 -3758.18,E2 -3758.18} C_VEL
LIN {X 0,Y 545.09,Z 142.083,A -85,B 0,C 180,E1 -3760.413,E2 -3760.413} C_VEL
LIN {X 0,Y 545.03,Z 142.089,A -85,B 0,C 180,E1 -3763.52,E2 -3763.52} C_VEL
LIN {X 0,Y 545.05,Z 142.085,A -85,B 0,C 180,E1 -3765.818,E2 -3765.818} C_VEL
LIN {X 0,Y 545.094,Z 142.088,A -85,B 0,C 180,E1 -3768.849,E2 -3768.849} C_VEL
LIN {X 0,Y 545.075,Z 142.083,A -85,B 0,C 180,E1 -3771.846,E2 -3771.846} C_VEL
LIN {X 0,Y 545.173,Z 142.077,A -85,B 0,C 180,E1 -3774.822,E2 -3774.822} C_VEL
LIN {X 0,Y 545.164,Z 142.072,A -85,B 0,C 180,E1 -3777.783,E2 -3777.783} C_VEL
LIN {X 0,Y 545.195,Z 142.075,A -85,B 0,C 180,E1 -3780.738,E2 -3780.738} C_VEL
LIN {X 0,Y 545.139,Z 142.077,A -85,B 0,C 180,E1 -3782.956,E2 -3782.956} C_VEL
LIN {X 0,Y 545.114,Z 142.08,A -85,B 0,C 180,E1 -3785.92,E2 -3785.92} C_VEL
LIN {X 0,Y 545.05,Z 142.092,A -85,B 0,C 180,E1 -3788.154,E2 -3788.154} C_VEL
LIN {X 0,Y 545.056,Z 142.086,A -85,B 0,C 180,E1 -3791.152,E2 -3791.152} C_VEL
LIN {X 0,Y 545.065,Z 142.092,A -85,B 0,C 180,E1 -3794.18,E2 -3794.18} C_VEL
LIN {X 0,Y 545.041,Z 142.088,A -85,B 0,C 180,E1 -3797.415,E2 -3797.415} C_VEL
LIN {X 0,Y 545.075,Z 142.091,A -85,B 0,C 180,E1 -3800.372,E2 -3800.372} C_VEL
LIN {X 0,Y 545.059,Z 142.087,A -85,B 0,C 180,E1 -3803.56,E2 -3803.56} C_VEL
LIN {X 0,Y 545.025,Z 142.097,A -85,B 0,C 180,E1 -3806.003,E2 -3806.003} C_VEL
LIN {X 0,Y 545.006,Z 142.095,A -85,B 0,C 180,E1 -3808.735,E2 -3808.735} C_VEL
LIN {X 0,Y 545.038,Z 142.091,A -85,B 0,C 180,E1 -3811.049,E2 -3811.049} C_VEL
LIN {X 0,Y 545.084,Z 142.13,A -85,B 0,C 180,E1 -3813.066,E2 -3813.066} C_VEL
LIN {X 0,Y 545.664,Z 146.197,A -85,B 0,C 180,E1 -3813.84,E2 -3813.84} C_VEL
LIN {X 0,Y 545.549,Z 156.038,A -85,B 0,C 180,E1 -3815.532,E2 -3815.532} C_VEL
LIN {X 0,Y 544.828,Z 159.199,A -85,B 0,C 180,E1 -3816.052,E2 -3816.052} C_VEL
LIN {X 0,Y 538.982,Z 169.904,A -85,B 0,C 180,E1 -3817.711,E2 -3817.711} C_VEL
LIN {X 0,Y 538.314,Z 173.064,A -85,B 0,C 180,E1 -3818.239,E2 -3818.239} C_VEL
LIN {X 0,Y 538.266,Z 179.26,A -85,B 0,C 180,E1 -3819.275,E2 -3819.275} C_VEL
LIN {X 0,Y 539.323,Z 185.652,A -85,B 0,C 180,E1 -3819.423,E2 -3819.423} C_VEL
LIN {X 0,Y 539.664,Z 190.339,A -85,B 0,C 180,E1 -3819.497,E2 -3819.497} C_VEL
LIN {X 0,Y 539.313,Z 287.172,A -85,B 0,C 180,E1 -3820.818,E2 -3820.818} C_VEL
LIN {X 0,Y 539.132,Z 299.92,A -85,B 0,C 180,E1 -3821.145,E2 -3821.145} C_VEL
LIN {X 0,Y 538.96,Z 311.541,A -85,B 0,C 180,E1 -3821.58,E2 -3821.58} C_VEL
LIN {X 0,Y 538.736,Z 323.087,A -85,B 0,C 180,E1 -3822.15,E2 -3822.15} C_VEL
LIN {X 0,Y 538.464,Z 335.58,A -85,B 0,C 180,E1 -3822.96,E2 -3822.96} C_VEL
LIN {X 0,Y 538.279,Z 345.624,A -85,B 0,C 180,E1 -3823.787,E2 -3823.787} C_VEL
LIN {X 0,Y 538.105,Z 352.959,A -85,B 0,C 180,E1 -3824.509,E2 -3824.509} C_VEL
LIN {X 0,Y 537.927,Z 360.235,A -85,B 0,C 180,E1 -3825.354,E2 -3825.354} C_VEL
LIN {X 0,Y 537.792,Z 366.184,A -85,B 0,C 180,E1 -3826.164,E2 -3826.164} C_VEL
LIN {X 0,Y 537.7,Z 372.439,A -85,B 0,C 180,E1 -3827.184,E2 -3827.184} C_VEL
LIN {X 0,Y 537.644,Z 377.504,A -85,B 0,C 180,E1 -3828.192,E2 -3828.192} C_VEL
LIN {X 0,Y 537.587,Z 382.003,A -85,B 0,C 180,E1 -3829.309,E2 -3829.309} C_VEL
LIN {X 0,Y 537.498,Z 385.6,A -85,B 0,C 180,E1 -3830.484,E2 -3830.484} C_VEL
LIN {X 0,Y 537.431,Z 388.177,A -85,B 0,C 180,E1 -3831.685,E2 -3831.685} C_VEL
LIN {X 0,Y 537.447,Z 389.784,A -85,B 0,C 180,E1 -3833.022,E2 -3833.022} C_VEL
LIN {X 0,Y 537.435,Z 390.139,A -85,B 0,C 180,E1 -3834.171,E2 -3834.171} C_VEL
LIN {X 0,Y 537.46,Z 389.395,A -85,B 0,C 180,E1 -3835.467,E2 -3835.467} C_VEL
LIN {X 0,Y 537.467,Z 387.378,A -85,B 0,C 180,E1 -3836.811,E2 -3836.811} C_VEL
LIN {X 0,Y 537.555,Z 383.972,A -85,B 0,C 180,E1 -3838.19,E2 -3838.19} C_VEL
LIN {X 0,Y 537.589,Z 378.695,A -85,B 0,C 180,E1 -3839.635,E2 -3839.635} C_VEL
LIN {X 0,Y 537.716,Z 373.825,A -85,B 0,C 180,E1 -3840.652,E2 -3840.652} C_VEL
LIN {X 0,Y 537.82,Z 367.416,A -85,B 0,C 180,E1 -3841.737,E2 -3841.737} C_VEL
LIN {X 0,Y 537.926,Z 360.708,A -85,B 0,C 180,E1 -3842.674,E2 -3842.674} C_VEL
LIN {X 0,Y 538.083,Z 352.434,A -85,B 0,C 180,E1 -3843.637,E2 -3843.637} C_VEL
LIN {X 0,Y 538.317,Z 342.488,A -85,B 0,C 180,E1 -3844.585,E2 -3844.585} C_VEL
LIN {X 0,Y 538.57,Z 331.621,A -85,B 0,C 180,E1 -3845.408,E2 -3845.408} C_VEL
LIN {X 0,Y 538.796,Z 321.277,A -85,B 0,C 180,E1 -3846.036,E2 -3846.036} C_VEL
LIN {X 0,Y 538.982,Z 310.205,A -85,B 0,C 180,E1 -3846.567,E2 -3846.567} C_VEL
LIN {X 0,Y 539.151,Z 297.984,A -85,B 0,C 180,E1 -3847.006,E2 -3847.006} C_VEL
LIN {X 0,Y 539.315,Z 284.741,A -85,B 0,C 180,E1 -3847.315,E2 -3847.315} C_VEL
LIN {X 0,Y 539.595,Z 187.327,A -85,B 0,C 180,E1 -3848.638,E2 -3848.638} C_VEL
LIN {X 0,Y 538.226,Z 179.439,A -85,B 0,C 180,E1 -3848.807,E2 -3848.807} C_VEL
LIN {X 0,Y 538.306,Z 174.884,A -85,B 0,C 180,E1 -3849.556,E2 -3849.556} C_VEL
LIN {X 0,Y 538.596,Z 158.107,A -85,B 0,C 180,E1 -3852.536,E2 -3852.536} C_VEL
LIN {X 0,Y 538.765,Z 147.233,A -85,B 0,C 180,E1 -3854.491,E2 -3854.491} C_VEL
LIN {X 0,Y 538.105,Z 142.989,A -85,B 0,C 180,E1 -3855.343,E2 -3855.343} C_VEL
LIN {X 0,Y 538.074,Z 142.958,A -85,B 0,C 180,E1 -3858.702,E2 -3858.702} C_VEL
LIN {X 0,Y 538.084,Z 142.96,A -85,B 0,C 180,E1 -3861.74,E2 -3861.74} C_VEL
LIN {X 0,Y 538.158,Z 142.944,A -85,B 0,C 180,E1 -3864.756,E2 -3864.756} C_VEL
LIN {X 0,Y 538.163,Z 142.953,A -85,B 0,C 180,E1 -3867.756,E2 -3867.756} C_VEL
LIN {X 0,Y 538.18,Z 142.942,A -85,B 0,C 180,E1 -3870.749,E2 -3870.749} C_VEL
LIN {X 0,Y 538.135,Z 142.948,A -85,B 0,C 180,E1 -3872.995,E2 -3872.995} C_VEL
LIN {X 0,Y 538.117,Z 142.953,A -85,B 0,C 180,E1 -3875.998,E2 -3875.998} C_VEL
LIN {X 0,Y 538.059,Z 142.959,A -85,B 0,C 180,E1 -3879.018,E2 -3879.018} C_VEL
LIN {X 0,Y 538.082,Z 142.956,A -85,B 0,C 180,E1 -3882.063,E2 -3882.063} C_VEL
LIN {X 0,Y 538.044,Z 142.964,A -85,B 0,C 180,E1 -3885.144,E2 -3885.144} C_VEL
LIN {X 0,Y 538.024,Z 142.961,A -85,B 0,C 180,E1 -3888.271,E2 -3888.271} C_VEL
LIN {X 0,Y 538.036,Z 142.961,A -85,B 0,C 180,E1 -3890.652,E2 -3890.652} C_VEL
LIN {X 0,Y 538.001,Z 142.965,A -85,B 0,C 180,E1 -3893.889,E2 -3893.889} C_VEL
LIN {X 0,Y 538.04,Z 142.959,A -85,B 0,C 180,E1 -3896.367,E2 -3896.367} C_VEL
LIN {X 0,Y 538.029,Z 142.967,A -85,B 0,C 180,E1 -3898.934,E2 -3898.934} C_VEL
LIN {X 0,Y 538.009,Z 142.963,A -85,B 0,C 180,E1 -3901.887,E2 -3901.887} C_VEL
LIN {X 0,Y 538.008,Z 142.967,A -85,B 0,C 180,E1 -3904.618,E2 -3904.618} C_VEL
LIN {X 0,Y 538.003,Z 142.969,A -85,B 0,C 180,E1 -3907.17,E2 -3907.17} C_VEL
LIN {X 0,Y 538.009,Z 142.963,A -85,B 0,C 180,E1 -3909.798,E2 -3909.798} C_VEL
LIN {X 0,Y 538.018,Z 142.971,A -85,B 0,C 180,E1 -3912.786,E2 -3912.786} C_VEL
LIN {X 0,Y 538.017,Z 142.962,A -85,B 0,C 180,E1 -3915.927,E2 -3915.927} C_VEL
LIN {X 0,Y 538.047,Z 142.96,A -85,B 0,C 180,E1 -3919.253,E2 -3919.253} C_VEL
LIN {X 0,Y 537.986,Z 142.968,A -85,B 0,C 180,E1 -3922.122,E2 -3922.122} C_VEL
LIN {X 0,Y 537.993,Z 142.969,A -85,B 0,C 180,E1 -3924.916,E2 -3924.916} C_VEL
LIN {X 0,Y 538.017,Z 142.962,A -85,B 0,C 180,E1 -3927.618,E2 -3927.618} C_VEL
LIN {X 0,Y 538.011,Z 142.969,A -85,B 0,C 180,E1 -3930.239,E2 -3930.239} C_VEL
LIN {X 0,Y 538.013,Z 142.966,A -85,B 0,C 180,E1 -3932.794,E2 -3932.794} C_VEL
LIN {X 0,Y 538.021,Z 142.961,A -85,B 0,C 180,E1 -3935.292,E2 -3935.292} C_VEL
LIN {X 0,Y 538.013,Z 142.968,A -85,B 0,C 180,E1 -3938.043,E2 -3938.043} C_VEL
LIN {X 0,Y 538.079,Z 142.963,A -85,B 0,C 180,E1 -3940.148,E2 -3940.148} C_VEL
LIN {X 0,Y 537.993,Z 142.965,A -85,B 0,C 180,E1 -3943.298,E2 -3943.298} C_VEL
LIN {X 0,Y 538.05,Z 142.961,A -85,B 0,C 180,E1 -3945.631,E2 -3945.631} C_VEL
LIN {X 0,Y 538.075,Z 142.956,A -85,B 0,C 180,E1 -3948.702,E2 -3948.702} C_VEL
LIN {X 0,Y 538.049,Z 142.964,A -85,B 0,C 180,E1 -3951.739,E2 -3951.739} C_VEL
LIN {X 0,Y 538.128,Z 142.948,A -85,B 0,C 180,E1 -3954.755,E2 -3954.755} C_VEL
LIN {X 0,Y 538.159,Z 142.953,A -85,B 0,C 180,E1 -3957.755,E2 -3957.755} C_VEL
LIN {X 0,Y 538.155,Z 142.951,A -85,B 0,C 180,E1 -3960,E2 -3960} C_VEL
LIN {X 0,Y 538.123,Z 142.949,A -85,B 0,C 180,E1 -3962.995,E2 -3962.995} C_VEL
LIN {X 0,Y 538.074,Z 142.959,A -85,B 0,C 180,E1 -3965.998,E2 -3965.998} C_VEL
LIN {X 0,Y 538.027,Z 142.962,A -85,B 0,C 180,E1 -3969.019,E2 -3969.019} C_VEL
LIN {X 0,Y 538.052,Z 142.96,A -85,B 0,C 180,E1 -3972.064,E2 -3972.064} C_VEL
LIN {X 0,Y 538.037,Z 142.964,A -85,B 0,C 180,E1 -3975.144,E2 -3975.144} C_VEL
LIN {X 0,Y 538.005,Z 142.963,A -85,B 0,C 180,E1 -3978.271,E2 -3978.271} C_VEL
LIN {X 0,Y 538.004,Z 142.965,A -85,B 0,C 180,E1 -3980.653,E2 -3980.653} C_VEL
LIN {X 0,Y 538.005,Z 142.97,A -85,B 0,C 180,E1 -3983.073,E2 -3983.073} C_VEL
LIN {X 0,Y 537.983,Z 142.969,A -85,B 0,C 180,E1 -3985.659,E2 -3985.659} C_VEL
LIN {X 0,Y 537.972,Z 142.968,A -85,B 0,C 180,E1 -3988.054,E2 -3988.054} C_VEL
LIN {X 0,Y 537.988,Z 142.968,A -85,B 0,C 180,E1 -3990.629,E2 -3990.629} C_VEL
LIN {X 0,Y 537.999,Z 142.97,A -85,B 0,C 180,E1 -3993.275,E2 -3993.275} C_VEL
LIN {X 0,Y 537.956,Z 142.969,A -85,B 0,C 180,E1 -3996.008,E2 -3996.008} C_VEL
LIN {X 0,Y 538,Z 142.972,A -85,B 0,C 180,E1 -3998.832,E2 -3998.832} C_VEL
LIN {X 0,Y 537.975,Z 142.967,A -85,B 0,C 180,E1 -4001.872,E2 -4001.872} C_VEL
LIN {X 0,Y 537.986,Z 142.974,A -85,B 0,C 180,E1 -4004.865,E2 -4004.865} C_VEL
LIN {X 0,Y 537.96,Z 142.972,A -85,B 0,C 180,E1 -4007.208,E2 -4007.208} C_VEL
LIN {X 0,Y 537.963,Z 142.971,A -85,B 0,C 180,E1 -4010.197,E2 -4010.197} C_VEL
LIN {X 0,Y 537.947,Z 142.974,A -85,B 0,C 180,E1 -4013.061,E2 -4013.061} C_VEL
LIN {X 0,Y 537.945,Z 142.972,A -85,B 0,C 180,E1 -4015.821,E2 -4015.821} C_VEL
LIN {X 0,Y 537.991,Z 142.975,A -85,B 0,C 180,E1 -4018.497,E2 -4018.497} C_VEL
LIN {X 0,Y 537.987,Z 142.969,A -85,B 0,C 180,E1 -4021.095,E2 -4021.095} C_VEL
LIN {X 0,Y 537.98,Z 142.968,A -85,B 0,C 180,E1 -4023.63,E2 -4023.63} C_VEL
LIN {X 0,Y 538.05,Z 143.165,A -85,B 0,C 180,E1 -4026.828,E2 -4026.828} C_VEL
LIN {X 0,Y 539.112,Z 149.223,A -85,B 0,C 180,E1 -4027.901,E2 -4027.901} C_VEL
LIN {X 0,Y 538.883,Z 161.367,A -85,B 0,C 180,E1 -4029.887,E2 -4029.887} C_VEL
LIN {X 0,Y 538.559,Z 179.009,A -85,B 0,C 180,E1 -4032.729,E2 -4032.729} C_VEL
LIN {X 0,Y 538.321,Z 194.763,A -85,B 0,C 180,E1 -4035.218,E2 -4035.218} C_VEL
LIN {X 0,Y 538.79,Z 198.06,A -85,B 0,C 180,E1 -4035.311,E2 -4035.311} C_VEL
LIN {X 0,Y 539.66,Z 205.004,A -85,B 0,C 180,E1 -4035.43,E2 -4035.43} C_VEL
LIN {X 0,Y 539.298,Z 303.323,A -85,B 0,C 180,E1 -4036.769,E2 -4036.769} C_VEL
LIN {X 0,Y 539.129,Z 316.369,A -85,B 0,C 180,E1 -4037.1,E2 -4037.1} C_VEL
LIN {X 0,Y 538.904,Z 328.977,A -85,B 0,C 180,E1 -4037.573,E2 -4037.573} C_VEL
LIN {X 0,Y 538.689,Z 341.17,A -85,B 0,C 180,E1 -4038.201,E2 -4038.201} C_VEL
LIN {X 0,Y 538.462,Z 353.106,A -85,B 0,C 180,E1 -4038.995,E2 -4038.995} C_VEL
LIN {X 0,Y 538.227,Z 363.32,A -85,B 0,C 180,E1 -4039.846,E2 -4039.846} C_VEL
LIN {X 0,Y 538.022,Z 372.5,A -85,B 0,C 180,E1 -4040.791,E2 -4040.791} C_VEL
LIN {X 0,Y 537.842,Z 381.439,A -85,B 0,C 180,E1 -4041.924,E2 -4041.924} C_VEL
LIN {X 0,Y 537.686,Z 388.632,A -85,B 0,C 180,E1 -4043.055,E2 -4043.055} C_VEL
LIN {X 0,Y 537.677,Z 395.181,A -85,B 0,C 180,E1 -4044.373,E2 -4044.373} C_VEL
LIN {X 0,Y 537.554,Z 399.509,A -85,B 0,C 180,E1 -4045.5,E2 -4045.5} C_VEL
LIN {X 0,Y 537.591,Z 401.801,A -85,B 0,C 180,E1 -4046.251,E2 -4046.251} C_VEL
LIN {X 0,Y 537.551,Z 403.658,A -85,B 0,C 180,E1 -4047.002,E2 -4047.002} C_VEL
LIN {X 0,Y 537.451,Z 406.042,A -85,B 0,C 180,E1 -4048.501,E2 -4048.501} C_VEL
LIN {X 0,Y 537.443,Z 406.865,A -85,B 0,C 180,E1 -4049.999,E2 -4049.999} C_VEL
LIN {X 0,Y 537.451,Z 406.045,A -85,B 0,C 180,E1 -4051.498,E2 -4051.498} C_VEL
LIN {X 0,Y 537.49,Z 405.053,A -85,B 0,C 180,E1 -4052.247,E2 -4052.247} C_VEL
LIN {X 0,Y 537.551,Z 403.662,A -85,B 0,C 180,E1 -4052.997,E2 -4052.997} C_VEL
LIN {X 0,Y 537.603,Z 400.734,A -85,B 0,C 180,E1 -4054.122,E2 -4054.122} C_VEL
LIN {X 0,Y 537.587,Z 396.768,A -85,B 0,C 180,E1 -4055.25,E2 -4055.25} C_VEL
LIN {X 0,Y 537.641,Z 391.909,A -85,B 0,C 180,E1 -4056.328,E2 -4056.328} C_VEL
LIN {X 0,Y 537.771,Z 385.233,A -85,B 0,C 180,E1 -4057.508,E2 -4057.508} C_VEL
LIN {X 0,Y 537.941,Z 377.21,A -85,B 0,C 180,E1 -4058.64,E2 -4058.64} C_VEL
LIN {X 0,Y 538.112,Z 369.028,A -85,B 0,C 180,E1 -4059.585,E2 -4059.585} C_VEL
LIN {X 0,Y 538.354,Z 359.047,A -85,B 0,C 180,E1 -4060.53,E2 -4060.53} C_VEL
LIN {X 0,Y 538.56,Z 349.19,A -85,B 0,C 180,E1 -4061.287,E2 -4061.287} C_VEL
LIN {X 0,Y 538.754,Z 338.027,A -85,B 0,C 180,E1 -4061.975,E2 -4061.975} C_VEL
LIN {X 0,Y 538.943,Z 325.567,A -85,B 0,C 180,E1 -4062.568,E2 -4062.568} C_VEL
LIN {X 0,Y 539.198,Z 312.408,A -85,B 0,C 180,E1 -4063.016,E2 -4063.016} C_VEL
LIN {X 0,Y 539.343,Z 299.203,A -85,B 0,C 180,E1 -4063.3,E2 -4063.3} C_VEL
LIN {X 0,Y 539.536,Z 203.004,A -85,B 0,C 180,E1 -4064.6,E2 -4064.6} C_VEL
LIN {X 0,Y 538.307,Z 194.843,A -85,B 0,C 180,E1 -4064.771,E2 -4064.771} C_VEL
LIN {X 0,Y 538.55,Z 177.592,A -85,B 0,C 180,E1 -4067.465,E2 -4067.465} C_VEL
LIN {X 0,Y 538.929,Z 157.956,A -85,B 0,C 180,E1 -4070.615,E2 -4070.615} C_VEL
LIN {X 0,Y 538.928,Z 148.114,A -85,B 0,C 180,E1 -4072.22,E2 -4072.22} C_VEL
LIN {X 0,Y 538.025,Z 143.022,A -85,B 0,C 180,E1 -4073.146,E2 -4073.146} C_VEL
LIN {X 0,Y 537.979,Z 142.97,A -85,B 0,C 180,E1 -4076.369,E2 -4076.369} C_VEL
LIN {X 0,Y 537.969,Z 142.971,A -85,B 0,C 180,E1 -4078.921,E2 -4078.921} C_VEL
LIN {X 0,Y 537.994,Z 142.97,A -85,B 0,C 180,E1 -4081.884,E2 -4081.884} C_VEL
LIN {X 0,Y 537.989,Z 142.967,A -85,B 0,C 180,E1 -4084.614,E2 -4084.614} C_VEL
LIN {X 0,Y 537.957,Z 142.973,A -85,B 0,C 180,E1 -4087.879,E2 -4087.879} C_VEL
LIN {X 0,Y 537.984,Z 142.968,A -85,B 0,C 180,E1 -4090.78,E2 -4090.78} C_VEL
LIN {X 0,Y 537.988,Z 142.966,A -85,B 0,C 180,E1 -4094.069,E2 -4094.069} C_VEL
LIN {X 0,Y 537.961,Z 142.975,A -85,B 0,C 180,E1 -4097.018,E2 -4097.018} C_VEL
LIN {X 0,Y 537.99,Z 142.966,A -85,B 0,C 180,E1 -4100.2,E2 -4100.2} C_VEL
LIN {X 0,Y 537.981,Z 142.973,A -85,B 0,C 180,E1 -4103.063,E2 -4103.063} C_VEL
LIN {X 0,Y 537.986,Z 142.966,A -85,B 0,C 180,E1 -4105.824,E2 -4105.824} C_VEL
LIN {X 0,Y 537.977,Z 142.969,A -85,B 0,C 180,E1 -4108.496,E2 -4108.496} C_VEL
LIN {X 0,Y 537.972,Z 142.976,A -85,B 0,C 180,E1 -4111.094,E2 -4111.094} C_VEL
LIN {X 0,Y 537.974,Z 142.969,A -85,B 0,C 180,E1 -4113.629,E2 -4113.629} C_VEL
LIN {X 0,Y 537.993,Z 142.965,A -85,B 0,C 180,E1 -4116.122,E2 -4116.122} C_VEL
LIN {X 0,Y 538.019,Z 142.964,A -85,B 0,C 180,E1 -4119.348,E2 -4119.348} C_VEL
LIN {X 0,Y 538.015,Z 142.966,A -85,B 0,C 180,E1 -4122.515,E2 -4122.515} C_VEL
LIN {X 0,Y 538.023,Z 142.961,A -85,B 0,C 180,E1 -4125.629,E2 -4125.629} C_VEL
LIN {X 0,Y 538.056,Z 142.964,A -85,B 0,C 180,E1 -4128.701,E2 -4128.701} C_VEL
LIN {X 0,Y 538.039,Z 142.959,A -85,B 0,C 180,E1 -4131.739,E2 -4131.739} C_VEL
LIN {X 0,Y 538.073,Z 142.956,A -85,B 0,C 180,E1 -4134.002,E2 -4134.002} C_VEL
LIN {X 0,Y 538.111,Z 142.954,A -85,B 0,C 180,E1 -4137.005,E2 -4137.005} C_VEL
LIN {X 0,Y 538.165,Z 142.95,A -85,B 0,C 180,E1 -4140.748,E2 -4140.748} C_VEL
LIN {X 0,Y 538.105,Z 142.953,A -85,B 0,C 180,E1 -4142.994,E2 -4142.994} C_VEL
LIN {X 0,Y 538.071,Z 142.958,A -85,B 0,C 180,E1 -4145.998,E2 -4145.998} C_VEL
LIN {X 0,Y 538.021,Z 142.969,A -85,B 0,C 180,E1 -4148.261,E2 -4148.261} C_VEL
LIN {X 0,Y 538.023,Z 142.962,A -85,B 0,C 180,E1 -4151.573,E2 -4151.573} C_VEL
LIN {X 0,Y 538.041,Z 142.962,A -85,B 0,C 180,E1 -4154.856,E2 -4154.856} C_VEL
LIN {X 0,Y 537.99,Z 142.975,A -85,B 0,C 180,E1 -4158.271,E2 -4158.271} C_VEL
LIN {X 0,Y 538.02,Z 142.966,A -85,B 0,C 180,E1 -4160.652,E2 -4160.652} C_VEL
LIN {X 0,Y 537.992,Z 142.971,A -85,B 0,C 180,E1 -4163.878,E2 -4163.878} C_VEL
LIN {X 0,Y 537.968,Z 142.975,A -85,B 0,C 180,E1 -4166.37,E2 -4166.37} C_VEL
LIN {X 0,Y 537.977,Z 142.97,A -85,B 0,C 180,E1 -4168.926,E2 -4168.926} C_VEL
LIN {X 0,Y 537.996,Z 142.974,A -85,B 0,C 180,E1 -4171.887,E2 -4171.887} C_VEL
LIN {X 0,Y 538.059,Z 143.106,A -85,B 0,C 180,E1 -4172.991,E2 -4172.991} C_VEL
LIN {X 0,Y 538.696,Z 148.014,A -85,B 0,C 180,E1 -4173.898,E2 -4173.898} C_VEL
LIN {X 0,Y 538.447,Z 165.298,A -85,B 0,C 180,E1 -4176.899,E2 -4176.899} C_VEL
LIN {X 0,Y 538.314,Z 173.064,A -85,B 0,C 180,E1 -4178.239,E2 -4178.239} C_VEL
LIN {X 0,Y 538.055,Z 175.495,A -85,B 0,C 180,E1 -4178.557,E2 -4178.557} C_VEL
LIN {X 0,Y 536.985,Z 180.17,A -85,B 0,C 180,E1 -4178.914,E2 -4178.914} C_VEL
LIN {X 0,Y 535.541,Z 185.491,A -85,B 0,C 180,E1 -4179.148,E2 -4179.148} C_VEL
LIN {X 0,Y 533.629,Z 193.4,A -85,B 0,C 180,E1 -4179.338,E2 -4179.338} C_VEL
LIN {X 0,Y 532.831,Z 199.523,A -85,B 0,C 180,E1 -4179.43,E2 -4179.43} C_VEL
LIN {X 0,Y 532.779,Z 201.583,A -85,B 0,C 180,E1 -4179.458,E2 -4179.458} C_VEL
LIN {X 0,Y 532.406,Z 287.14,A -85,B 0,C 180,E1 -4180.644,E2 -4180.644} C_VEL
LIN {X 0,Y 532.22,Z 300.507,A -85,B 0,C 180,E1 -4180.993,E2 -4180.993} C_VEL
LIN {X 0,Y 532.023,Z 312.735,A -85,B 0,C 180,E1 -4181.463,E2 -4181.463} C_VEL
LIN {X 0,Y 531.731,Z 325.443,A -85,B 0,C 180,E1 -4182.126,E2 -4182.126} C_VEL
LIN {X 0,Y 531.455,Z 337.109,A -85,B 0,C 180,E1 -4182.924,E2 -4182.924} C_VEL
LIN {X 0,Y 531.254,Z 346.906,A -85,B 0,C 180,E1 -4183.761,E2 -4183.761} C_VEL
LIN {X 0,Y 531.008,Z 356.241,A -85,B 0,C 180,E1 -4184.732,E2 -4184.732} C_VEL
LIN {X 0,Y 530.794,Z 364.919,A -85,B 0,C 180,E1 -4185.851,E2 -4185.851} C_VEL
LIN {X 0,Y 530.672,Z 371.716,A -85,B 0,C 180,E1 -4186.94,E2 -4186.94} C_VEL
LIN {X 0,Y 530.57,Z 376.588,A -85,B 0,C 180,E1 -4187.883,E2 -4187.883} C_VEL
LIN {X 0,Y 530.527,Z 381.356,A -85,B 0,C 180,E1 -4189.033,E2 -4189.033} C_VEL
LIN {X 0,Y 530.416,Z 385.124,A -85,B 0,C 180,E1 -4190.219,E2 -4190.219} C_VEL
LIN {X 0,Y 530.33,Z 387.957,A -85,B 0,C 180,E1 -4191.477,E2 -4191.477} C_VEL
LIN {X 0,Y 530.34,Z 389.588,A -85,B 0,C 180,E1 -4192.665,E2 -4192.665} C_VEL
LIN {X 0,Y 530.329,Z 390.254,A -85,B 0,C 180,E1 -4193.937,E2 -4193.937} C_VEL
LIN {X 0,Y 530.372,Z 389.751,A -85,B 0,C 180,E1 -4195.266,E2 -4195.266} C_VEL
LIN {X 0,Y 530.36,Z 387.975,A -85,B 0,C 180,E1 -4196.598,E2 -4196.598} C_VEL
LIN {X 0,Y 530.454,Z 384.796,A -85,B 0,C 180,E1 -4197.987,E2 -4197.987} C_VEL
LIN {X 0,Y 530.484,Z 381.943,A -85,B 0,C 180,E1 -4198.891,E2 -4198.891} C_VEL
LIN {X 0,Y 530.52,Z 378.509,A -85,B 0,C 180,E1 -4199.776,E2 -4199.776} C_VEL
LIN {X 0,Y 530.666,Z 372.867,A -85,B 0,C 180,E1 -4200.936,E2 -4200.936} C_VEL
LIN {X 0,Y 530.768,Z 366.714,A -85,B 0,C 180,E1 -4201.963,E2 -4201.963} C_VEL
LIN {X 0,Y 530.945,Z 358.847,A -85,B 0,C 180,E1 -4203.042,E2 -4203.042} C_VEL
LIN {X 0,Y 531.215,Z 348.334,A -85,B 0,C 180,E1 -4204.194,E2 -4204.194} C_VEL
LIN {X 0,Y 531.432,Z 338.305,A -85,B 0,C 180,E1 -4205.07,E2 -4205.07} C_VEL
LIN {X 0,Y 531.702,Z 326.851,A -85,B 0,C 180,E1 -4205.877,E2 -4205.877} C_VEL
LIN {X 0,Y 531.982,Z 314.472,A -85,B 0,C 180,E1 -4206.549,E2 -4206.549} C_VEL
LIN {X 0,Y 532.175,Z 302.039,A -85,B 0,C 180,E1 -4207.047,E2 -4207.047} C_VEL
LIN {X 0,Y 532.334,Z 289.993,A -85,B 0,C 180,E1 -4207.388,E2 -4207.388} C_VEL
LIN {X 0,Y 532.464,Z 271.469,A -85,B 0,C 180,E1 -4207.682,E2 -4207.682} C_VEL
LIN {X 0,Y 532.675,Z 187.63,A -85,B 0,C 180,E1 -4208.829,E2 -4208.829} C_VEL
LIN {X 0,Y 531.239,Z 179.667,A -85,B 0,C 180,E1 -4208.997,E2 -4208.997} C_VEL
LIN {X 0,Y 531.248,Z 177.716,A -85,B 0,C 180,E1 -4209.276,E2 -4209.276} C_VEL
LIN {X 0,Y 531.603,Z 161.693,A -85,B 0,C 180,E1 -4212.15,E2 -4212.15} C_VEL
LIN {X 0,Y 531.829,Z 148.859,A -85,B 0,C 180,E1 -4214.48,E2 -4214.48} C_VEL
LIN {X 0,Y 531.065,Z 143.918,A -85,B 0,C 180,E1 -4215.463,E2 -4215.463} C_VEL
LIN {X 0,Y 531.034,Z 143.837,A -85,B 0,C 180,E1 -4218.551,E2 -4218.551} C_VEL
LIN {X 0,Y 531.053,Z 143.835,A -85,B 0,C 180,E1 -4221.63,E2 -4221.63} C_VEL
LIN {X 0,Y 531.117,Z 143.822,A -85,B 0,C 180,E1 -4224.686,E2 -4224.686} C_VEL
LIN {X 0,Y 531.135,Z 143.828,A -85,B 0,C 180,E1 -4227.726,E2 -4227.726} C_VEL
LIN {X 0,Y 531.15,Z 143.817,A -85,B 0,C 180,E1 -4230.759,E2 -4230.759} C_VEL
LIN {X 0,Y 531.102,Z 143.825,A -85,B 0,C 180,E1 -4233.035,E2 -4233.035} C_VEL
LIN {X 0,Y 531.073,Z 143.83,A -85,B 0,C 180,E1 -4236.078,E2 -4236.078} C_VEL
LIN {X 0,Y 531.021,Z 143.837,A -85,B 0,C 180,E1 -4239.139,E2 -4239.139} C_VEL
LIN {X 0,Y 531.039,Z 143.832,A -85,B 0,C 180,E1 -4242.226,E2 -4242.226} C_VEL
LIN {X 0,Y 530.994,Z 143.845,A -85,B 0,C 180,E1 -4245.35,E2 -4245.35} C_VEL
LIN {X 0,Y 530.984,Z 143.838,A -85,B 0,C 180,E1 -4248.522,E2 -4248.522} C_VEL
LIN {X 0,Y 530.998,Z 143.84,A -85,B 0,C 180,E1 -4250.938,E2 -4250.938} C_VEL
LIN {X 0,Y 530.963,Z 143.841,A -85,B 0,C 180,E1 -4254.226,E2 -4254.226} C_VEL
LIN {X 0,Y 531,Z 143.839,A -85,B 0,C 180,E1 -4256.744,E2 -4256.744} C_VEL
LIN {X 0,Y 530.979,Z 143.845,A -85,B 0,C 180,E1 -4259.323,E2 -4259.323} C_VEL
LIN {X 0,Y 530.964,Z 143.841,A -85,B 0,C 180,E1 -4262.101,E2 -4262.101} C_VEL
LIN {X 0,Y 530.967,Z 143.847,A -85,B 0,C 180,E1 -4264.851,E2 -4264.851} C_VEL
LIN {X 0,Y 530.964,Z 143.842,A -85,B 0,C 180,E1 -4267.508,E2 -4267.508} C_VEL
LIN {X 0,Y 530.976,Z 143.842,A -85,B 0,C 180,E1 -4270.434,E2 -4270.434} C_VEL
LIN {X 0,Y 530.959,Z 143.844,A -85,B 0,C 180,E1 -4273.281,E2 -4273.281} C_VEL
LIN {X 0,Y 530.976,Z 143.839,A -85,B 0,C 180,E1 -4275.622,E2 -4275.622} C_VEL
LIN {X 0,Y 530.988,Z 143.845,A -85,B 0,C 180,E1 -4278.564,E2 -4278.564} C_VEL
LIN {X 0,Y 530.952,Z 143.842,A -85,B 0,C 180,E1 -4281.529,E2 -4281.529} C_VEL
LIN {X 0,Y 530.948,Z 143.849,A -85,B 0,C 180,E1 -4284.38,E2 -4284.38} C_VEL
LIN {X 0,Y 530.966,Z 143.842,A -85,B 0,C 180,E1 -4287.134,E2 -4287.134} C_VEL
LIN {X 0,Y 530.959,Z 143.842,A -85,B 0,C 180,E1 -4289.803,E2 -4289.803} C_VEL
LIN {X 0,Y 530.965,Z 143.848,A -85,B 0,C 180,E1 -4292.478,E2 -4292.478} C_VEL
LIN {X 0,Y 530.985,Z 143.839,A -85,B 0,C 180,E1 -4294.942,E2 -4294.942} C_VEL
LIN {X 0,Y 530.969,Z 143.849,A -85,B 0,C 180,E1 -4298.247,E2 -4298.247} C_VEL
LIN {X 0,Y 530.98,Z 143.841,A -85,B 0,C 180,E1 -4300.677,E2 -4300.677} C_VEL
LIN {X 0,Y 530.957,Z 143.841,A -85,B 0,C 180,E1 -4303.07,E2 -4303.07} C_VEL
LIN {X 0,Y 531.007,Z 143.836,A -85,B 0,C 180,E1 -4305.436,E2 -4305.436} C_VEL
LIN {X 0,Y 531.033,Z 143.834,A -85,B 0,C 180,E1 -4308.55,E2 -4308.55} C_VEL
LIN {X 0,Y 530.998,Z 143.84,A -85,B 0,C 180,E1 -4311.629,E2 -4311.629} C_VEL
LIN {X 0,Y 531.088,Z 143.826,A -85,B 0,C 180,E1 -4314.685,E2 -4314.685} C_VEL
LIN {X 0,Y 531.131,Z 143.827,A -85,B 0,C 180,E1 -4317.725,E2 -4317.725} C_VEL
LIN {X 0,Y 531.124,Z 143.827,A -85,B 0,C 180,E1 -4320,E2 -4320} C_VEL
LIN {X 0,Y 531.091,Z 143.826,A -85,B 0,C 180,E1 -4323.035,E2 -4323.035} C_VEL
LIN {X 0,Y 531.033,Z 143.835,A -85,B 0,C 180,E1 -4326.078,E2 -4326.078} C_VEL
LIN {X 0,Y 530.993,Z 143.84,A -85,B 0,C 180,E1 -4329.139,E2 -4329.139} C_VEL
LIN {X 0,Y 531.047,Z 143.837,A -85,B 0,C 180,E1 -4331.669,E2 -4331.669} C_VEL
LIN {X 0,Y 531.018,Z 143.836,A -85,B 0,C 180,E1 -4334.95,E2 -4334.95} C_VEL
LIN {X 0,Y 530.972,Z 143.844,A -85,B 0,C 180,E1 -4337.724,E2 -4337.724} C_VEL
LIN {X 0,Y 531.009,Z 143.835,A -85,B 0,C 180,E1 -4340.128,E2 -4340.128} C_VEL
LIN {X 0,Y 530.94,Z 143.844,A -85,B 0,C 180,E1 -4342.574,E2 -4342.574} C_VEL
LIN {X 0,Y 530.939,Z 143.85,A -85,B 0,C 180,E1 -4345.061,E2 -4345.061} C_VEL
LIN {X 0,Y 530.951,Z 143.845,A -85,B 0,C 180,E1 -4347.599,E2 -4347.599} C_VEL
LIN {X 0,Y 530.942,Z 143.846,A -85,B 0,C 180,E1 -4350.639,E2 -4350.639} C_VEL
LIN {X 0,Y 530.947,Z 143.846,A -85,B 0,C 180,E1 -4353.497,E2 -4353.497} C_VEL
LIN {X 0,Y 530.903,Z 143.848,A -85,B 0,C 180,E1 -4356.147,E2 -4356.147} C_VEL
LIN {X 0,Y 530.955,Z 143.846,A -85,B 0,C 180,E1 -4358.652,E2 -4358.652} C_VEL
LIN {X 0,Y 530.909,Z 143.849,A -85,B 0,C 180,E1 -4361.444,E2 -4361.444} C_VEL
LIN {X 0,Y 530.96,Z 143.846,A -85,B 0,C 180,E1 -4364.55,E2 -4364.55} C_VEL
LIN {X 0,Y 530.905,Z 143.848,A -85,B 0,C 180,E1 -4367.536,E2 -4367.536} C_VEL
LIN {X 0,Y 530.929,Z 143.852,A -85,B 0,C 180,E1 -4370.551,E2 -4370.551} C_VEL
LIN {X 0,Y 530.896,Z 143.849,A -85,B 0,C 180,E1 -4373.436,E2 -4373.436} C_VEL
LIN {X 0,Y 530.941,Z 143.852,A -85,B 0,C 180,E1 -4376.504,E2 -4376.504} C_VEL
LIN {X 0,Y 530.944,Z 143.845,A -85,B 0,C 180,E1 -4379.361,E2 -4379.361} C_VEL
LIN {X 0,Y 530.955,Z 143.851,A -85,B 0,C 180,E1 -4382.48,E2 -4382.48} C_VEL
LIN {X 0,Y 530.949,Z 143.85,A -85,B 0,C 180,E1 -4385.774,E2 -4385.774} C_VEL
LIN {X 0,Y 530.971,Z 143.889,A -85,B 0,C 180,E1 -4386.604,E2 -4386.604} C_VEL
LIN {X 0,Y 531.597,Z 147.23,A -85,B 0,C 180,E1 -4387.25,E2 -4387.25} C_VEL
LIN {X 0,Y 532.171,Z 151.354,A -85,B 0,C 180,E1 -4387.968,E2 -4387.968} C_VEL
LIN {X 0,Y 531.811,Z 165.502,A -85,B 0,C 180,E1 -4390.306,E2 -4390.306} C_VEL
LIN {X 0,Y 531.524,Z 181.339,A -85,B 0,C 180,E1 -4392.89,E2 -4392.89} C_VEL
LIN {X 0,Y 531.309,Z 194.892,A -85,B 0,C 180,E1 -4395.035,E2 -4395.035} C_VEL
LIN {X 0,Y 532.802,Z 204.742,A -85,B 0,C 180,E1 -4395.236,E2 -4395.236} C_VEL
LIN {X 0,Y 532.4,Z 303.078,A -85,B 0,C 180,E1 -4396.594,E2 -4396.594} C_VEL
LIN {X 0,Y 532.22,Z 316.166,A -85,B 0,C 180,E1 -4396.93,E2 -4396.93} C_VEL
LIN {X 0,Y 531.983,Z 328.798,A -85,B 0,C 180,E1 -4397.409,E2 -4397.409} C_VEL
LIN {X 0,Y 531.735,Z 340.778,A -85,B 0,C 180,E1 -4398.03,E2 -4398.03} C_VEL
LIN {X 0,Y 531.471,Z 352.957,A -85,B 0,C 180,E1 -4398.848,E2 -4398.848} C_VEL
LIN {X 0,Y 531.225,Z 363.182,A -85,B 0,C 180,E1 -4399.711,E2 -4399.711} C_VEL
LIN {X 0,Y 530.979,Z 372.368,A -85,B 0,C 180,E1 -4400.668,E2 -4400.668} C_VEL
LIN {X 0,Y 530.775,Z 381.312,A -85,B 0,C 180,E1 -4401.816,E2 -4401.816} C_VEL
LIN {X 0,Y 530.625,Z 388.511,A -85,B 0,C 180,E1 -4402.962,E2 -4402.962} C_VEL
LIN {X 0,Y 530.591,Z 395.063,A -85,B 0,C 180,E1 -4404.298,E2 -4404.298} C_VEL
LIN {X 0,Y 530.452,Z 399.394,A -85,B 0,C 180,E1 -4405.44,E2 -4405.44} C_VEL
LIN {X 0,Y 530.516,Z 401.688,A -85,B 0,C 180,E1 -4406.201,E2 -4406.201} C_VEL
LIN {X 0,Y 530.457,Z 403.546,A -85,B 0,C 180,E1 -4406.961,E2 -4406.961} C_VEL
LIN {X 0,Y 530.411,Z 404.939,A -85,B 0,C 180,E1 -4407.721,E2 -4407.721} C_VEL
LIN {X 0,Y 530.345,Z 406.539,A -85,B 0,C 180,E1 -4409.24,E2 -4409.24} C_VEL
LIN {X 0,Y 530.344,Z 406.755,A -85,B 0,C 180,E1 -4409.999,E2 -4409.999} C_VEL
LIN {X 0,Y 530.361,Z 405.933,A -85,B 0,C 180,E1 -4411.518,E2 -4411.518} C_VEL
LIN {X 0,Y 530.411,Z 404.941,A -85,B 0,C 180,E1 -4412.277,E2 -4412.277} C_VEL
LIN {X 0,Y 530.457,Z 403.548,A -85,B 0,C 180,E1 -4413.037,E2 -4413.037} C_VEL
LIN {X 0,Y 530.522,Z 400.618,A -85,B 0,C 180,E1 -4414.177,E2 -4414.177} C_VEL
LIN {X 0,Y 530.524,Z 396.648,A -85,B 0,C 180,E1 -4415.32,E2 -4415.32} C_VEL
LIN {X 0,Y 530.594,Z 390.952,A -85,B 0,C 180,E1 -4416.577,E2 -4416.577} C_VEL
LIN {X 0,Y 530.708,Z 383.867,A -85,B 0,C 180,E1 -4417.8,E2 -4417.8} C_VEL
LIN {X 0,Y 530.898,Z 375.58,A -85,B 0,C 180,E1 -4418.948,E2 -4418.948} C_VEL
LIN {X 0,Y 531.077,Z 367.078,A -85,B 0,C 180,E1 -4419.905,E2 -4419.905} C_VEL
LIN {X 0,Y 531.383,Z 356.571,A -85,B 0,C 180,E1 -4420.862,E2 -4420.862} C_VEL
LIN {X 0,Y 531.64,Z 345.681,A -85,B 0,C 180,E1 -4421.662,E2 -4421.662} C_VEL
LIN {X 0,Y 531.872,Z 334.753,A -85,B 0,C 180,E1 -4422.301,E2 -4422.301} C_VEL
LIN {X 0,Y 532.111,Z 322.988,A -85,B 0,C 180,E1 -4422.829,E2 -4422.829} C_VEL
LIN {X 0,Y 532.285,Z 309.419,A -85,B 0,C 180,E1 -4423.261,E2 -4423.261} C_VEL
LIN {X 0,Y 532.456,Z 295.756,A -85,B 0,C 180,E1 -4423.524,E2 -4423.524} C_VEL
LIN {X 0,Y 532.765,Z 204.344,A -85,B 0,C 180,E1 -4424.769,E2 -4424.769} C_VEL
LIN {X 0,Y 531.277,Z 194.846,A -85,B 0,C 180,E1 -4424.962,E2 -4424.962} C_VEL
LIN {X 0,Y 531.447,Z 183.599,A -85,B 0,C 180,E1 -4426.715,E2 -4426.715} C_VEL
LIN {X 0,Y 531.743,Z 167.648,A -85,B 0,C 180,E1 -4429.293,E2 -4429.293} C_VEL
LIN {X 0,Y 532.118,Z 150.995,A -85,B 0,C 180,E1 -4432.019,E2 -4432.019} C_VEL
LIN {X 0,Y 530.97,Z 143.924,A -85,B 0,C 180,E1 -4433.292,E2 -4433.292} C_VEL
LIN {X 0,Y 530.959,Z 143.849,A -85,B 0,C 180,E1 -4435.899,E2 -4435.899} C_VEL
LIN {X 0,Y 530.925,Z 143.848,A -85,B 0,C 180,E1 -4438.458,E2 -4438.458} C_VEL
LIN {X 0,Y 530.932,Z 143.849,A -85,B 0,C 180,E1 -4441.079,E2 -4441.079} C_VEL
LIN {X 0,Y 530.944,Z 143.85,A -85,B 0,C 180,E1 -4443.774,E2 -4443.774} C_VEL
LIN {X 0,Y 530.899,Z 143.85,A -85,B 0,C 180,E1 -4446.561,E2 -4446.561} C_VEL
LIN {X 0,Y 530.939,Z 143.852,A -85,B 0,C 180,E1 -4449.446,E2 -4449.446} C_VEL
LIN {X 0,Y 530.897,Z 143.85,A -85,B 0,C 180,E1 -4452.463,E2 -4452.463} C_VEL
LIN {X 0,Y 530.952,Z 143.85,A -85,B 0,C 180,E1 -4455.449,E2 -4455.449} C_VEL
LIN {X 0,Y 530.943,Z 143.845,A -85,B 0,C 180,E1 -4458.559,E2 -4458.559} C_VEL
LIN {X 0,Y 530.937,Z 143.848,A -85,B 0,C 180,E1 -4461.527,E2 -4461.527} C_VEL
LIN {X 0,Y 530.936,Z 143.845,A -85,B 0,C 180,E1 -4464.378,E2 -4464.378} C_VEL
LIN {X 0,Y 530.942,Z 143.853,A -85,B 0,C 180,E1 -4467.131,E2 -4467.131} C_VEL
LIN {X 0,Y 530.922,Z 143.846,A -85,B 0,C 180,E1 -4469.8,E2 -4469.8} C_VEL
LIN {X 0,Y 530.95,Z 143.844,A -85,B 0,C 180,E1 -4472.477,E2 -4472.477} C_VEL
LIN {X 0,Y 530.933,Z 143.854,A -85,B 0,C 180,E1 -4474.938,E2 -4474.938} C_VEL
LIN {X 0,Y 530.963,Z 143.841,A -85,B 0,C 180,E1 -4477.898,E2 -4477.898} C_VEL
LIN {X 0,Y 530.958,Z 143.847,A -85,B 0,C 180,E1 -4480.676,E2 -4480.676} C_VEL
LIN {X 0,Y 530.945,Z 143.848,A -85,B 0,C 180,E1 -4483.069,E2 -4483.069} C_VEL
LIN {X 0,Y 530.984,Z 143.839,A -85,B 0,C 180,E1 -4485.435,E2 -4485.435} C_VEL
LIN {X 0,Y 531.016,Z 143.84,A -85,B 0,C 180,E1 -4488.549,E2 -4488.549} C_VEL
LIN {X 0,Y 531.015,Z 143.834,A -85,B 0,C 180,E1 -4491.628,E2 -4491.628} C_VEL
LIN {X 0,Y 531.088,Z 143.834,A -85,B 0,C 180,E1 -4494.685,E2 -4494.685} C_VEL
LIN {X 0,Y 531.111,Z 143.822,A -85,B 0,C 180,E1 -4497.725,E2 -4497.725} C_VEL
LIN {X 0,Y 531.135,Z 143.826,A -85,B 0,C 180,E1 -4500.758,E2 -4500.758} C_VEL
LIN {X 0,Y 531.071,Z 143.828,A -85,B 0,C 180,E1 -4503.034,E2 -4503.034} C_VEL
LIN {X 0,Y 531.032,Z 143.836,A -85,B 0,C 180,E1 -4506.077,E2 -4506.077} C_VEL
LIN {X 0,Y 530.972,Z 143.849,A -85,B 0,C 180,E1 -4508.371,E2 -4508.371} C_VEL
LIN {X 0,Y 530.995,Z 143.838,A -85,B 0,C 180,E1 -4511.65,E2 -4511.65} C_VEL
LIN {X 0,Y 531.013,Z 143.837,A -85,B 0,C 180,E1 -4514.955,E2 -4514.955} C_VEL
LIN {X 0,Y 530.956,Z 143.845,A -85,B 0,C 180,E1 -4517.724,E2 -4517.724} C_VEL
LIN {X 0,Y 531.01,Z 143.843,A -85,B 0,C 180,E1 -4520.127,E2 -4520.127} C_VEL
LIN {X 0,Y 530.928,Z 143.85,A -85,B 0,C 180,E1 -4522.574,E2 -4522.574} C_VEL
LIN {X 0,Y 530.935,Z 143.845,A -85,B 0,C 180,E1 -4525.061,E2 -4525.061} C_VEL
LIN {X 0,Y 530.936,Z 143.848,A -85,B 0,C 180,E1 -4527.599,E2 -4527.599} C_VEL
LIN {X 0,Y 530.941,Z 143.849,A -85,B 0,C 180,E1 -4530.642,E2 -4530.642} C_VEL
LIN {X 0,Y 531.029,Z 143.971,A -85,B 0,C 180,E1 -4532.862,E2 -4532.862} C_VEL
LIN {X 0,Y 531.715,Z 149.808,A -85,B 0,C 180,E1 -4533.948,E2 -4533.948} C_VEL
LIN {X 0,Y 531.439,Z 167.199,A -85,B 0,C 180,E1 -4536.992,E2 -4536.992} C_VEL
LIN {X 0,Y 531.236,Z 179.328,A -85,B 0,C 180,E1 -4539.073,E2 -4539.073} C_VEL
LIN {X 0,Y 532.211,Z 184.837,A -85,B 0,C 180,E1 -4539.21,E2 -4539.21} C_VEL
LIN {X 0,Y 532.799,Z 190.559,A -85,B 0,C 180,E1 -4539.307,E2 -4539.307} C_VEL
LIN {X 0,Y 532.779,Z 201.583,A -85,B 0,C 180,E1 -4539.458,E2 -4539.458} C_VEL
LIN {X 0,Y 532.173,Z 207.422,A -85,B 0,C 180,E1 -4539.521,E2 -4539.521} C_VEL
LIN {X 0,Y 526.54,Z 226.417,A -85,B 0,C 180,E1 -4539.628,E2 -4539.628} C_VEL
LIN {X 0,Y 525.754,Z 232.261,A -85,B 0,C 180,E1 -4539.688,E2 -4539.688} C_VEL
LIN {X 0,Y 525.491,Z 287.617,A -85,B 0,C 180,E1 -4540.476,E2 -4540.476} C_VEL
LIN {X 0,Y 525.303,Z 301.033,A -85,B 0,C 180,E1 -4540.834,E2 -4540.834} C_VEL
LIN {X 0,Y 525.091,Z 313.432,A -85,B 0,C 180,E1 -4541.323,E2 -4541.323} C_VEL
LIN {X 0,Y 524.759,Z 326.675,A -85,B 0,C 180,E1 -4542.039,E2 -4542.039} C_VEL
LIN {X 0,Y 524.474,Z 337.494,A -85,B 0,C 180,E1 -4542.798,E2 -4542.798} C_VEL
LIN {X 0,Y 524.253,Z 347.026,A -85,B 0,C 180,E1 -4543.624,E2 -4543.624} C_VEL
LIN {X 0,Y 523.984,Z 357.081,A -85,B 0,C 180,E1 -4544.696,E2 -4544.696} C_VEL
LIN {X 0,Y 523.755,Z 365.108,A -85,B 0,C 180,E1 -4545.754,E2 -4545.754} C_VEL
LIN {X 0,Y 523.607,Z 371.612,A -85,B 0,C 180,E1 -4546.803,E2 -4546.803} C_VEL
LIN {X 0,Y 523.49,Z 377.952,A -85,B 0,C 180,E1 -4548.082,E2 -4548.082} C_VEL
LIN {X 0,Y 523.43,Z 382.899,A -85,B 0,C 180,E1 -4549.37,E2 -4549.37} C_VEL
LIN {X 0,Y 523.287,Z 386.966,A -85,B 0,C 180,E1 -4550.861,E2 -4550.861} C_VEL
LIN {X 0,Y 523.219,Z 388.745,A -85,B 0,C 180,E1 -4551.84,E2 -4551.84} C_VEL
LIN {X 0,Y 523.239,Z 389.873,A -85,B 0,C 180,E1 -4552.814,E2 -4552.814} C_VEL
LIN {X 0,Y 523.233,Z 390.332,A -85,B 0,C 180,E1 -4553.774,E2 -4553.774} C_VEL
LIN {X 0,Y 523.265,Z 390.048,A -85,B 0,C 180,E1 -4555.013,E2 -4555.013} C_VEL
LIN {X 0,Y 523.276,Z 388.172,A -85,B 0,C 180,E1 -4556.589,E2 -4556.589} C_VEL
LIN {X 0,Y 523.363,Z 385.62,A -85,B 0,C 180,E1 -4557.778,E2 -4557.778} C_VEL
LIN {X 0,Y 523.404,Z 382.39,A -85,B 0,C 180,E1 -4558.863,E2 -4558.863} C_VEL
LIN {X 0,Y 523.499,Z 377.009,A -85,B 0,C 180,E1 -4560.218,E2 -4560.218} C_VEL
LIN {X 0,Y 523.62,Z 370.112,A -85,B 0,C 180,E1 -4561.546,E2 -4561.546} C_VEL
LIN {X 0,Y 523.831,Z 362.265,A -85,B 0,C 180,E1 -4562.729,E2 -4562.729} C_VEL
LIN {X 0,Y 524.03,Z 354.092,A -85,B 0,C 180,E1 -4563.733,E2 -4563.733} C_VEL
LIN {X 0,Y 524.307,Z 344.41,A -85,B 0,C 180,E1 -4564.707,E2 -4564.707} C_VEL
LIN {X 0,Y 524.608,Z 332.842,A -85,B 0,C 180,E1 -4565.639,E2 -4565.639} C_VEL
LIN {X 0,Y 524.882,Z 322.139,A -85,B 0,C 180,E1 -4566.317,E2 -4566.317} C_VEL
LIN {X 0,Y 525.116,Z 310.312,A -85,B 0,C 180,E1 -4566.903,E2 -4566.903} C_VEL
LIN {X 0,Y 525.314,Z 298.355,A -85,B 0,C 180,E1 -4567.343,E2 -4567.343} C_VEL
LIN {X 0,Y 525.524,Z 285,A -85,B 0,C 180,E1 -4567.664,E2 -4567.664} C_VEL
LIN {X 0,Y 525.838,Z 188.455,A -85,B 0,C 180,E1 -4569.015,E2 -4569.015} C_VEL
LIN {X 0,Y 524.264,Z 179.798,A -85,B 0,C 180,E1 -4569.2,E2 -4569.2} C_VEL
LIN {X 0,Y 524.248,Z 178.777,A -85,B 0,C 180,E1 -4569.316,E2 -4569.316} C_VEL
LIN {X 0,Y 524.621,Z 162.544,A -85,B 0,C 180,E1 -4572.257,E2 -4572.257} C_VEL
LIN {X 0,Y 524.83,Z 149.747,A -85,B 0,C 180,E1 -4574.611,E2 -4574.611} C_VEL
LIN {X 0,Y 524.021,Z 144.793,A -85,B 0,C 180,E1 -4575.61,E2 -4575.61} C_VEL
LIN {X 0,Y 524.009,Z 144.714,A -85,B 0,C 180,E1 -4578.395,E2 -4578.395} C_VEL
LIN {X 0,Y 524.002,Z 144.712,A -85,B 0,C 180,E1 -4581.517,E2 -4581.517} C_VEL
LIN {X 0,Y 524.079,Z 144.699,A -85,B 0,C 180,E1 -4584.615,E2 -4584.615} C_VEL
LIN {X 0,Y 524.108,Z 144.702,A -85,B 0,C 180,E1 -4587.695,E2 -4587.695} C_VEL
LIN {X 0,Y 524.12,Z 144.693,A -85,B 0,C 180,E1 -4590.769,E2 -4590.769} C_VEL
LIN {X 0,Y 524.069,Z 144.701,A -85,B 0,C 180,E1 -4593.076,E2 -4593.076} C_VEL
LIN {X 0,Y 524.035,Z 144.706,A -85,B 0,C 180,E1 -4596.16,E2 -4596.16} C_VEL
LIN {X 0,Y 523.991,Z 144.714,A -85,B 0,C 180,E1 -4599.263,E2 -4599.263} C_VEL
LIN {X 0,Y 524.001,Z 144.713,A -85,B 0,C 180,E1 -4601.74,E2 -4601.74} C_VEL
LIN {X 0,Y 523.992,Z 144.713,A -85,B 0,C 180,E1 -4605.053,E2 -4605.053} C_VEL
LIN {X 0,Y 523.946,Z 144.716,A -85,B 0,C 180,E1 -4607.97,E2 -4607.97} C_VEL
LIN {X 0,Y 523.971,Z 144.712,A -85,B 0,C 180,E1 -4610.411,E2 -4610.411} C_VEL
LIN {X 0,Y 523.91,Z 144.723,A -85,B 0,C 180,E1 -4612.894,E2 -4612.894} C_VEL
LIN {X 0,Y 523.982,Z 144.711,A -85,B 0,C 180,E1 -4616.02,E2 -4616.02} C_VEL
LIN {X 0,Y 523.928,Z 144.723,A -85,B 0,C 180,E1 -4618.876,E2 -4618.876} C_VEL
LIN {X 0,Y 523.918,Z 144.721,A -85,B 0,C 180,E1 -4621.545,E2 -4621.545} C_VEL
LIN {X 0,Y 523.919,Z 144.719,A -85,B 0,C 180,E1 -4624.292,E2 -4624.292} C_VEL
LIN {X 0,Y 523.906,Z 144.726,A -85,B 0,C 180,E1 -4627.133,E2 -4627.133} C_VEL
LIN {X 0,Y 523.937,Z 144.717,A -85,B 0,C 180,E1 -4630.13,E2 -4630.13} C_VEL
LIN {X 0,Y 523.934,Z 144.72,A -85,B 0,C 180,E1 -4632.459,E2 -4632.459} C_VEL
LIN {X 0,Y 523.944,Z 144.717,A -85,B 0,C 180,E1 -4635.31,E2 -4635.31} C_VEL
LIN {X 0,Y 523.951,Z 144.724,A -85,B 0,C 180,E1 -4638.691,E2 -4638.691} C_VEL
LIN {X 0,Y 523.914,Z 144.722,A -85,B 0,C 180,E1 -4641.081,E2 -4641.081} C_VEL
LIN {X 0,Y 523.893,Z 144.722,A -85,B 0,C 180,E1 -4643.825,E2 -4643.825} C_VEL
LIN {X 0,Y 523.94,Z 144.723,A -85,B 0,C 180,E1 -4646.636,E2 -4646.636} C_VEL
LIN {X 0,Y 523.948,Z 144.715,A -85,B 0,C 180,E1 -4649.356,E2 -4649.356} C_VEL
LIN {X 0,Y 523.94,Z 144.723,A -85,B 0,C 180,E1 -4652.289,E2 -4652.289} C_VEL
LIN {X 0,Y 523.92,Z 144.718,A -85,B 0,C 180,E1 -4655.428,E2 -4655.428} C_VEL
LIN {X 0,Y 523.943,Z 144.717,A -85,B 0,C 180,E1 -4658.767,E2 -4658.767} C_VEL
LIN {X 0,Y 523.935,Z 144.716,A -85,B 0,C 180,E1 -4661.221,E2 -4661.221} C_VEL
LIN {X 0,Y 523.915,Z 144.721,A -85,B 0,C 180,E1 -4663.639,E2 -4663.639} C_VEL
LIN {X 0,Y 523.925,Z 144.726,A -85,B 0,C 180,E1 -4666.028,E2 -4666.028} C_VEL
LIN {X 0,Y 524.013,Z 144.71,A -85,B 0,C 180,E1 -4668.394,E2 -4668.394} C_VEL
LIN {X 0,Y 523.96,Z 144.716,A -85,B 0,C 180,E1 -4671.516,E2 -4671.516} C_VEL
LIN {X 0,Y 524.035,Z 144.705,A -85,B 0,C 180,E1 -4674.614,E2 -4674.614} C_VEL
LIN {X 0,Y 524.102,Z 144.702,A -85,B 0,C 180,E1 -4677.695,E2 -4677.695} C_VEL
LIN {X 0,Y 524.093,Z 144.702,A -85,B 0,C 180,E1 -4680,E2 -4680} C_VEL
LIN {X 0,Y 524.033,Z 144.705,A -85,B 0,C 180,E1 -4683.075,E2 -4683.075} C_VEL
LIN {X 0,Y 523.996,Z 144.711,A -85,B 0,C 180,E1 -4686.16,E2 -4686.16} C_VEL
LIN {X 0,Y 523.946,Z 144.719,A -85,B 0,C 180,E1 -4689.263,E2 -4689.263} C_VEL
LIN {X 0,Y 523.995,Z 144.715,A -85,B 0,C 180,E1 -4691.735,E2 -4691.735} C_VEL
LIN {X 0,Y 523.982,Z 144.714,A -85,B 0,C 180,E1 -4695.048,E2 -4695.048} C_VEL
LIN {X 0,Y 523.914,Z 144.72,A -85,B 0,C 180,E1 -4697.971,E2 -4697.971} C_VEL
LIN {X 0,Y 523.944,Z 144.715,A -85,B 0,C 180,E1 -4700.412,E2 -4700.412} C_VEL
LIN {X 0,Y 523.906,Z 144.723,A -85,B 0,C 180,E1 -4702.894,E2 -4702.894} C_VEL
LIN {X 0,Y 523.878,Z 144.729,A -85,B 0,C 180,E1 -4705.423,E2 -4705.423} C_VEL
LIN {X 0,Y 523.896,Z 144.721,A -85,B 0,C 180,E1 -4708.004,E2 -4708.004} C_VEL
LIN {X 0,Y 523.898,Z 144.726,A -85,B 0,C 180,E1 -4710.846,E2 -4710.846} C_VEL
LIN {X 0,Y 523.913,Z 144.72,A -85,B 0,C 180,E1 -4713.727,E2 -4713.727} C_VEL
LIN {X 0,Y 523.861,Z 144.727,A -85,B 0,C 180,E1 -4716.395,E2 -4716.395} C_VEL
LIN {X 0,Y 523.902,Z 144.727,A -85,B 0,C 180,E1 -4719.087,E2 -4719.087} C_VEL
LIN {X 0,Y 523.887,Z 144.723,A -85,B 0,C 180,E1 -4722.126,E2 -4722.126} C_VEL
LIN {X 0,Y 523.931,Z 144.719,A -85,B 0,C 180,E1 -4725.312,E2 -4725.312} C_VEL
LIN {X 0,Y 523.878,Z 144.732,A -85,B 0,C 180,E1 -4728.7,E2 -4728.7} C_VEL
LIN {X 0,Y 523.872,Z 144.725,A -85,B 0,C 180,E1 -4731.894,E2 -4731.894} C_VEL
LIN {X 0,Y 523.865,Z 144.729,A -85,B 0,C 180,E1 -4734.921,E2 -4734.921} C_VEL
LIN {X 0,Y 523.9,Z 144.721,A -85,B 0,C 180,E1 -4737.686,E2 -4737.686} C_VEL
LIN {X 0,Y 523.868,Z 144.732,A -85,B 0,C 180,E1 -4740.239,E2 -4740.239} C_VEL
LIN {X 0,Y 523.893,Z 144.725,A -85,B 0,C 180,E1 -4742.863,E2 -4742.863} C_VEL
LIN {X 0,Y 523.913,Z 144.727,A -85,B 0,C 180,E1 -4745.809,E2 -4745.809} C_VEL
LIN {X 0,Y 523.949,Z 144.866,A -85,B 0,C 180,E1 -4746.481,E2 -4746.481} C_VEL
LIN {X 0,Y 525.162,Z 151.746,A -85,B 0,C 180,E1 -4747.74,E2 -4747.74} C_VEL
LIN {X 0,Y 524.923,Z 164.19,A -85,B 0,C 180,E1 -4749.833,E2 -4749.833} C_VEL
LIN {X 0,Y 524.528,Z 181.236,A -85,B 0,C 180,E1 -4752.655,E2 -4752.655} C_VEL
LIN {X 0,Y 524.285,Z 194.799,A -85,B 0,C 180,E1 -4754.831,E2 -4754.831} C_VEL
LIN {X 0,Y 525.946,Z 205.404,A -85,B 0,C 180,E1 -4755.05,E2 -4755.05} C_VEL
LIN {X 0,Y 525.509,Z 302.833,A -85,B 0,C 180,E1 -4756.415,E2 -4756.415} C_VEL
LIN {X 0,Y 525.319,Z 315.963,A -85,B 0,C 180,E1 -4756.755,E2 -4756.755} C_VEL
LIN {X 0,Y 525.029,Z 328.618,A -85,B 0,C 180,E1 -4757.239,E2 -4757.239} C_VEL
LIN {X 0,Y 524.799,Z 340.332,A -85,B 0,C 180,E1 -4757.852,E2 -4757.852} C_VEL
LIN {X 0,Y 524.531,Z 351.514,A -85,B 0,C 180,E1 -4758.601,E2 -4758.601} C_VEL
LIN {X 0,Y 524.232,Z 361.988,A -85,B 0,C 180,E1 -4759.475,E2 -4759.475} C_VEL
